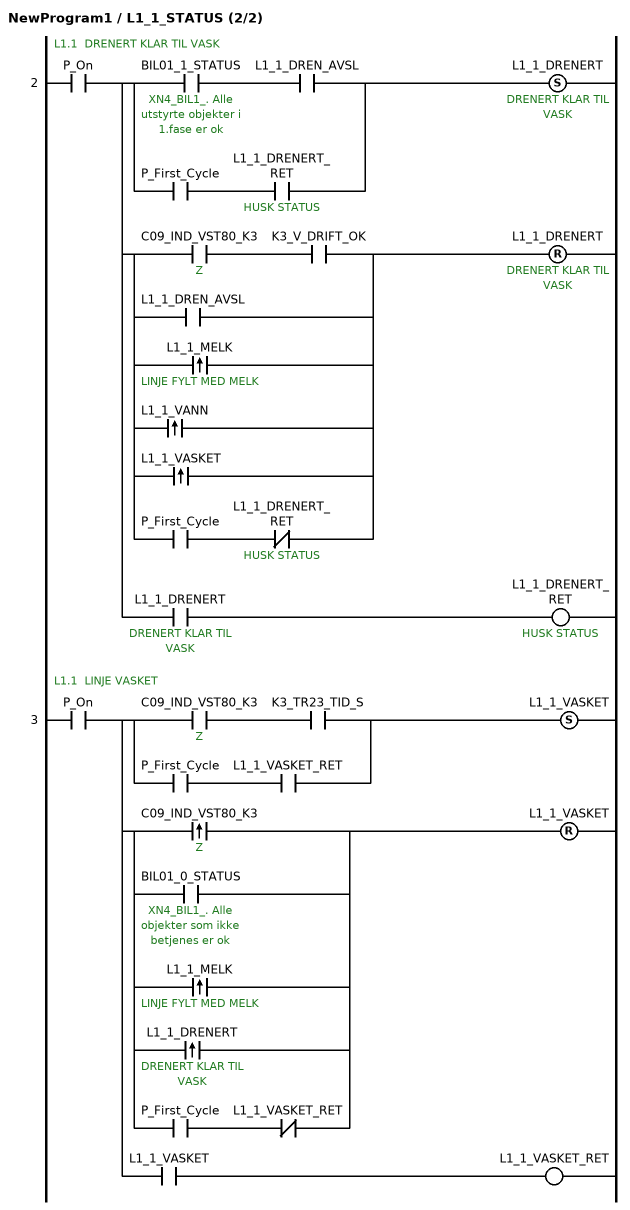
; [picture p768: NewProgram1 / L1_1_STATUS, rungs 2-3]
; rung 2: L1.1  DRENERT KLAR TIL VASK
LD P_On
OUT TR0
LD BIL01_1_STATUS  ; XN4_BIL1_. Alle utstyrte objekter i 1.fase er ok
AND L1_1_DREN_AVSL
LD P_First_Cycle
AND L1_1_DRENERT_RET  ; HUSK STATUS
ORLD
ANDLD
SET L1_1_DRENERT  ; DRENERT KLAR TIL VASK
LD TR0
LD C09_IND_VST80_K3  ; Z
AND K3_V_DRIFT_OK
OR L1_1_DREN_AVSL
@OR L1_1_MELK  ; LINJE FYLT MED MELK
@OR L1_1_VANN
@OR L1_1_VASKET
LD P_First_Cycle
ANDNOT L1_1_DRENERT_RET  ; HUSK STATUS
ORLD
ANDLD
RSET L1_1_DRENERT  ; DRENERT KLAR TIL VASK
LD TR0
AND L1_1_DRENERT  ; DRENERT KLAR TIL VASK
OUT L1_1_DRENERT_RET  ; HUSK STATUS
; rung 3: L1.1  LINJE VASKET
LD P_On
OUT TR0
LD C09_IND_VST80_K3  ; Z
AND K3_TR23_TID_S
LD P_First_Cycle
AND L1_1_VASKET_RET
ORLD
ANDLD
SET L1_1_VASKET
LD TR0
@LD C09_IND_VST80_K3  ; Z
OR BIL01_0_STATUS  ; XN4_BIL1_. Alle objekter som ikke betjenes er ok
@OR L1_1_MELK  ; LINJE FYLT MED MELK
@OR L1_1_DRENERT  ; DRENERT KLAR TIL VASK
LD P_First_Cycle
ANDNOT L1_1_VASKET_RET
ORLD
ANDLD
RSET L1_1_VASKET
LD TR0
AND L1_1_VASKET
OUT L1_1_VASKET_RET
; rung 4: Ingen_kommentar_funnet

### Section L1_1_FUNKSJONER

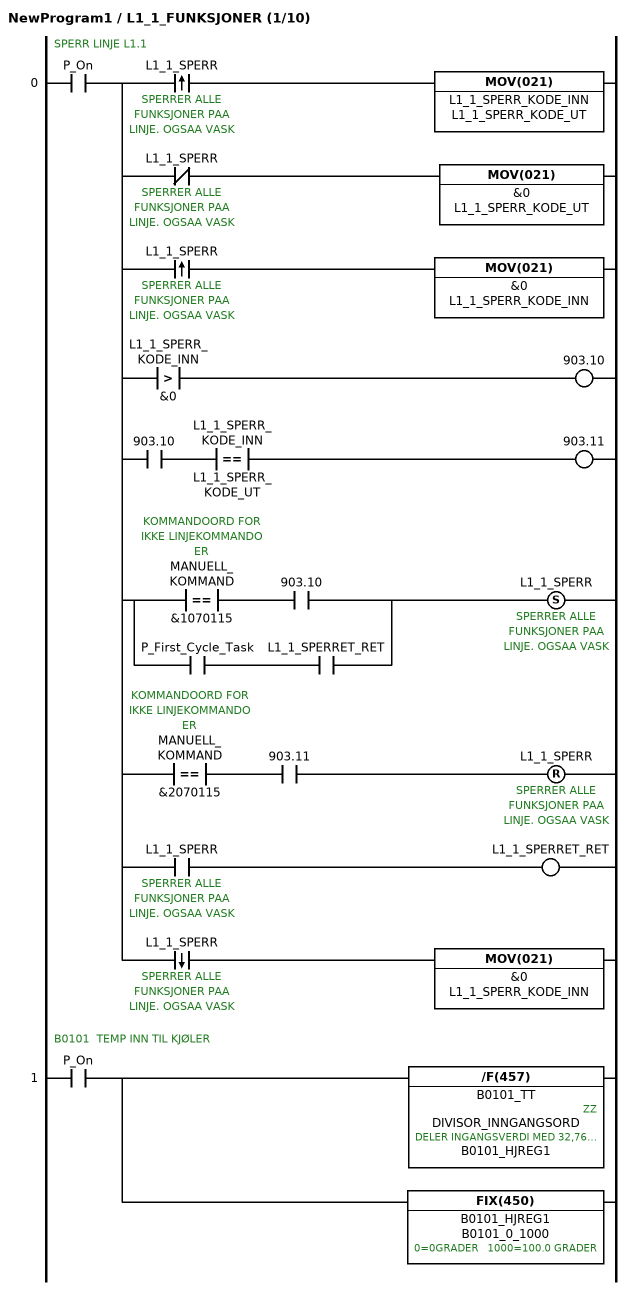
; rung 0: SPERR LINJE L1.1
LD P_On
OUT TR0
@AND L1_1_SPERR  ; SPERRER ALLE FUNKSJONER PAA LINJE. OGSAA VASK
MOV(021) L1_1_SPERR_KODE_INN L1_1_SPERR_KODE_UT
LD TR0
ANDNOT L1_1_SPERR  ; SPERRER ALLE FUNKSJONER PAA LINJE. OGSAA VASK
MOV(021) &0 L1_1_SPERR_KODE_UT
LD TR0
@AND L1_1_SPERR  ; SPERRER ALLE FUNKSJONER PAA LINJE. OGSAA VASK
MOV(021) &0 L1_1_SPERR_KODE_INN
LD TR0
AND>(320) L1_1_SPERR_KODE_INN &0
OUT 903.10
LD TR0
AND 903.10
AND=(300) L1_1_SPERR_KODE_INN L1_1_SPERR_KODE_UT
OUT 903.11
LD TR0
LD=L(301) MANUELL_KOMMAND &1070115  ; KOMMANDOORD FOR IKKE LINJEKOMMANDOER
AND 903.10
LD P_First_Cycle_Task
AND L1_1_SPERRET_RET
ORLD
ANDLD
SET L1_1_SPERR  ; SPERRER ALLE FUNKSJONER PAA LINJE. OGSAA VASK
LD TR0
AND=L(301) MANUELL_KOMMAND &2070115  ; KOMMANDOORD FOR IKKE LINJEKOMMANDOER
AND 903.11
RSET L1_1_SPERR  ; SPERRER ALLE FUNKSJONER PAA LINJE. OGSAA VASK
LD TR0
AND L1_1_SPERR  ; SPERRER ALLE FUNKSJONER PAA LINJE. OGSAA VASK
OUT L1_1_SPERRET_RET
LD TR0
%AND L1_1_SPERR  ; SPERRER ALLE FUNKSJONER PAA LINJE. OGSAA VASK
MOV(021) &0 L1_1_SPERR_KODE_INN
; rung 1: B0101  TEMP INN TIL KJØLER
LD P_On
/F(457) B0101_TT DIVISOR_INNGANGSORD B0101_HJREG1  ; ZZ, DELER INGANGSVERDI MED 32,760 FOR OMREGNING TIL 0-1000
FIX(450) B0101_HJREG1 B0101_0_1000  ; 0=0GRADER   1000=100.0 GRADER

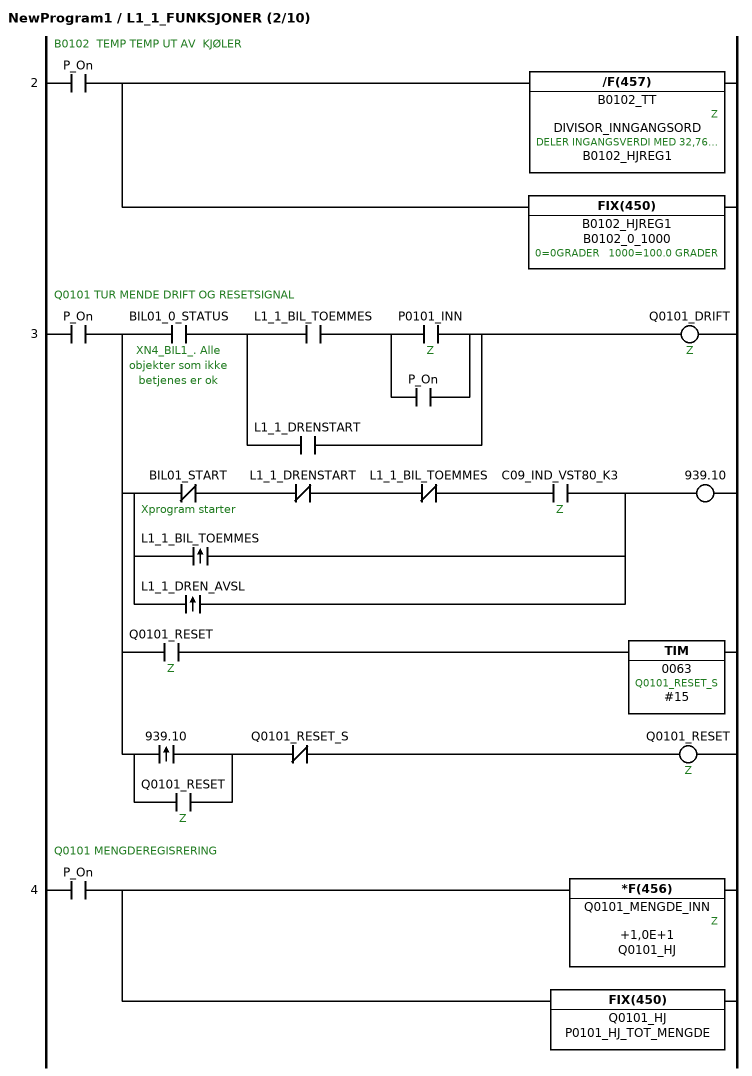
; rung 2: B0102  TEMP TEMP UT AV  KJØLER
LD P_On
/F(457) B0102_TT DIVISOR_INNGANGSORD B0102_HJREG1  ; Z, DELER INGANGSVERDI MED 32,760 FOR OMREGNING TIL 0-1000
FIX(450) B0102_HJREG1 B0102_0_1000  ; 0=0GRADER   1000=100.0 GRADER
; rung 3: Q0101 TUR MENDE DRIFT OG RESETSIGNAL
LD P_On
OUT TR0
AND BIL01_0_STATUS  ; XN4_BIL1_. Alle objekter som ikke betjenes er ok
LD L1_1_BIL_TOEMMES
LD P0101_INN  ; Z
OR P_On
ANDLD
OR L1_1_DRENSTART
ANDLD
OUT Q0101_DRIFT  ; Z
LD TR0
LDNOT BIL01_START  ; Xprogram starter
ANDNOT L1_1_DRENSTART
ANDNOT L1_1_BIL_TOEMMES
AND C09_IND_VST80_K3  ; Z
@OR L1_1_BIL_TOEMMES
@OR L1_1_DREN_AVSL
ANDLD
OUT 939.10
LD TR0
AND Q0101_RESET  ; Z
TIM 0063 #15  ; Q0101_RESET_S
LD TR0
@LD 939.10
OR Q0101_RESET  ; Z
ANDLD
ANDNOT Q0101_RESET_S
OUT Q0101_RESET  ; Z
; rung 4: Q0101 MENGDEREGISRERING
LD P_On
*F(456) Q0101_MENGDE_INN +1,0E+1 Q0101_HJ  ; Z
FIX(450) Q0101_HJ P0101_HJ_TOT_MENGDE

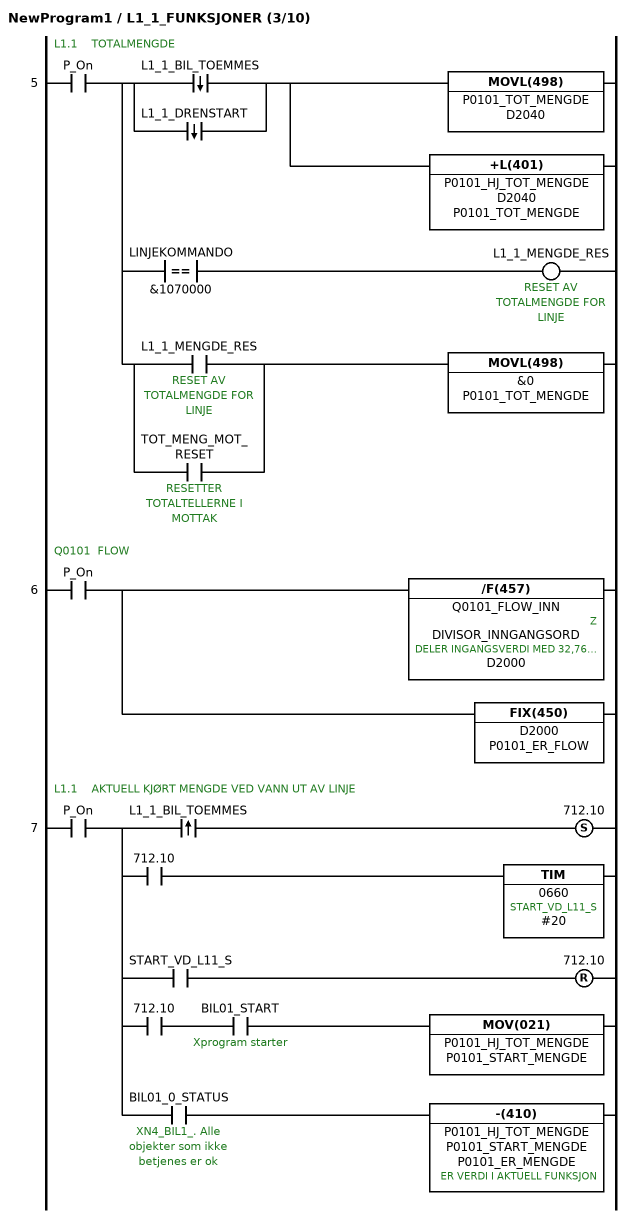
; rung 5: L1.1    TOTALMENGDE
LD P_On
OUT TR0
%LD L1_1_BIL_TOEMMES
%OR L1_1_DRENSTART
ANDLD
MOVL(498) P0101_TOT_MENGDE D2040
+L(401) P0101_HJ_TOT_MENGDE D2040 P0101_TOT_MENGDE
LD TR0
AND=L(301) LINJEKOMMANDO &1070000
OUT L1_1_MENGDE_RES  ; RESET AV  TOTALMENGDE FOR LINJE
LD TR0
LD L1_1_MENGDE_RES  ; RESET AV  TOTALMENGDE FOR LINJE
OR TOT_MENG_MOT_RESET  ; RESETTER TOTALTELLERNE I MOTTAK
ANDLD
MOVL(498) &0 P0101_TOT_MENGDE
; rung 6: Q0101  FLOW
LD P_On
/F(457) Q0101_FLOW_INN DIVISOR_INNGANGSORD D2000  ; Z, DELER INGANGSVERDI MED 32,760 FOR OMREGNING TIL 0-1000
FIX(450) D2000 P0101_ER_FLOW
; rung 7: L1.1    AKTUELL KJØRT MENGDE VED VANN UT AV LINJE
LD P_On
OUT TR0
@AND L1_1_BIL_TOEMMES
SET 712.10
LD TR0
AND 712.10
TIM 0660 #20  ; START_VD_L11_S
LD TR0
AND START_VD_L11_S
RSET 712.10
LD TR0
AND 712.10
AND BIL01_START  ; Xprogram starter
MOV(021) P0101_HJ_TOT_MENGDE P0101_START_MENGDE
LD TR0
AND BIL01_0_STATUS  ; XN4_BIL1_. Alle objekter som ikke betjenes er ok
-(410) P0101_HJ_TOT_MENGDE P0101_START_MENGDE P0101_ER_MENGDE  ; ER VERDI I AKTUELL FUNKSJON

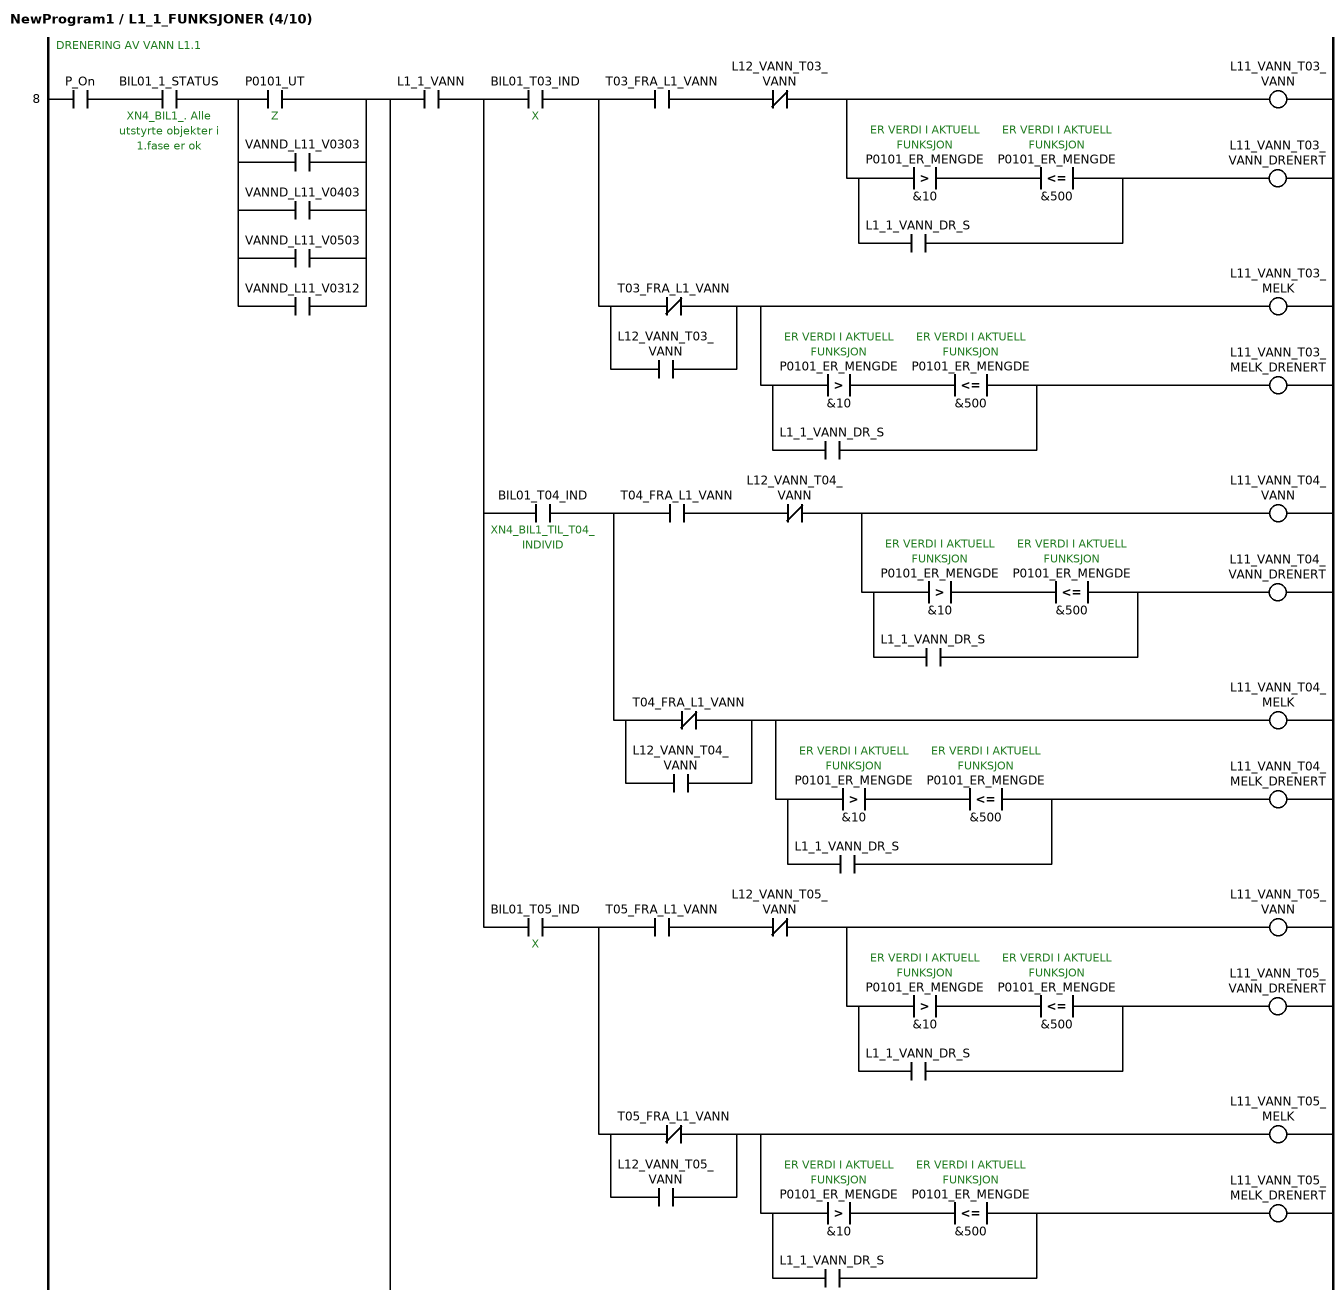

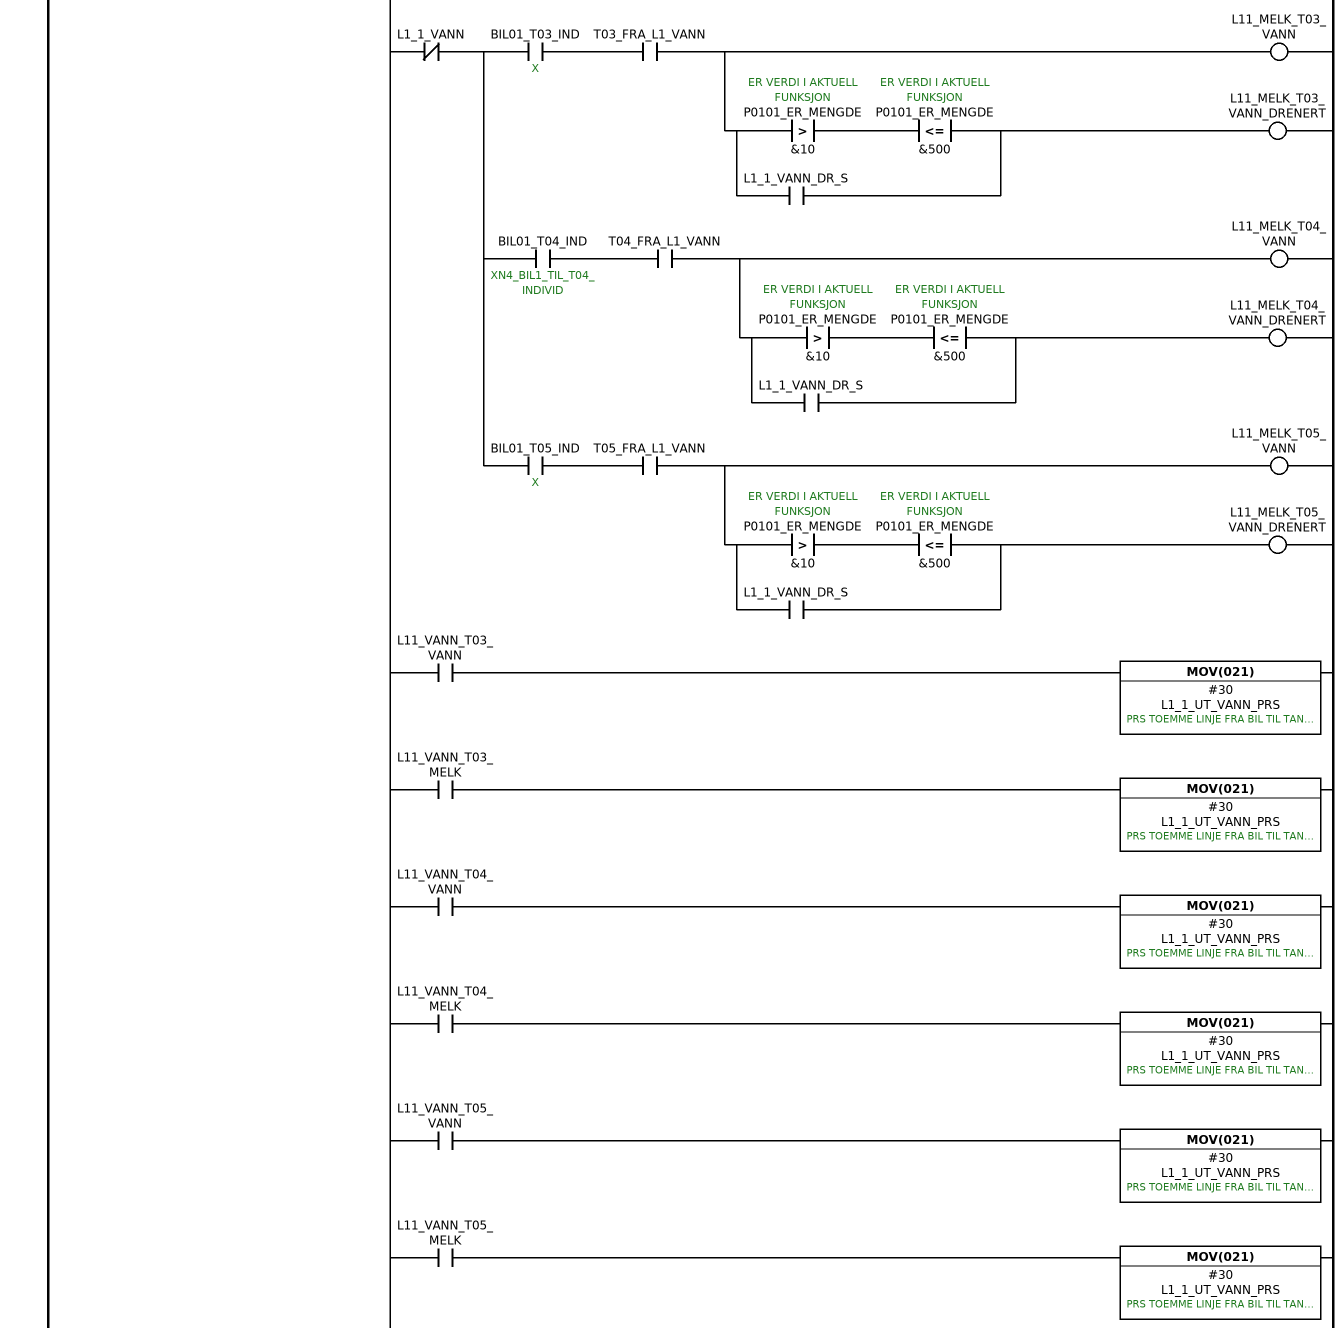

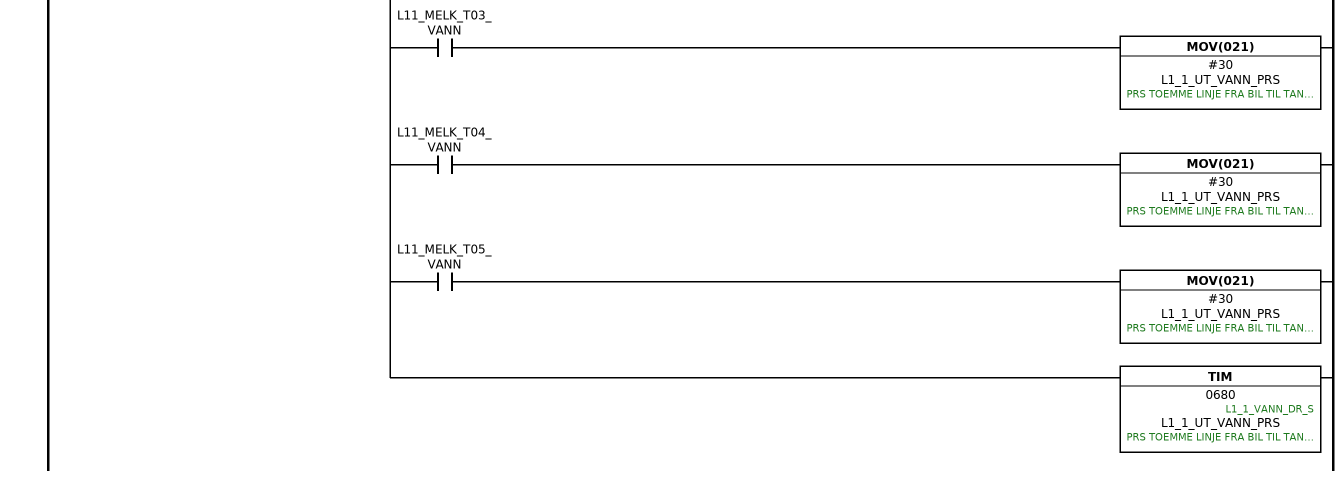
; rung 8: DRENERING AV VANN L1.1
LD P_On
AND BIL01_1_STATUS  ; XN4_BIL1_. Alle utstyrte objekter i 1.fase er ok
LD P0101_UT  ; Z
OR VANND_L11_V0303
OR VANND_L11_V0403
OR VANND_L11_V0503
OR VANND_L11_V0312
ANDLD
OUT TR0
AND L1_1_VANN
OUT TR1
AND BIL01_T03_IND  ; X
OUT TR2
AND T03_FRA_L1_VANN
ANDNOT L12_VANN_T03_VANN
OUT L11_VANN_T03_VANN
LD>(320) P0101_ER_MENGDE &10  ; ER VERDI I AKTUELL FUNKSJON
AND<=(315) P0101_ER_MENGDE &500  ; ER VERDI I AKTUELL FUNKSJON
OR L1_1_VANN_DR_S
ANDLD
OUT L11_VANN_T03_VANN_DRENERT
LD TR2
LDNOT T03_FRA_L1_VANN
OR L12_VANN_T03_VANN
ANDLD
OUT L11_VANN_T03_MELK
LD>(320) P0101_ER_MENGDE &10  ; ER VERDI I AKTUELL FUNKSJON
AND<=(315) P0101_ER_MENGDE &500  ; ER VERDI I AKTUELL FUNKSJON
OR L1_1_VANN_DR_S
ANDLD
OUT L11_VANN_T03_MELK_DRENERT
LD TR1
AND BIL01_T04_IND  ; XN4_BIL1_TIL_T04_INDIVID
OUT TR2
AND T04_FRA_L1_VANN
ANDNOT L12_VANN_T04_VANN
OUT L11_VANN_T04_VANN
LD>(320) P0101_ER_MENGDE &10  ; ER VERDI I AKTUELL FUNKSJON
AND<=(315) P0101_ER_MENGDE &500  ; ER VERDI I AKTUELL FUNKSJON
OR L1_1_VANN_DR_S
ANDLD
OUT L11_VANN_T04_VANN_DRENERT
LD TR2
LDNOT T04_FRA_L1_VANN
OR L12_VANN_T04_VANN
ANDLD
OUT L11_VANN_T04_MELK
LD>(320) P0101_ER_MENGDE &10  ; ER VERDI I AKTUELL FUNKSJON
AND<=(315) P0101_ER_MENGDE &500  ; ER VERDI I AKTUELL FUNKSJON
OR L1_1_VANN_DR_S
ANDLD
OUT L11_VANN_T04_MELK_DRENERT
LD TR1
AND BIL01_T05_IND  ; X
OUT TR1
AND T05_FRA_L1_VANN
ANDNOT L12_VANN_T05_VANN
OUT L11_VANN_T05_VANN
LD>(320) P0101_ER_MENGDE &10  ; ER VERDI I AKTUELL FUNKSJON
AND<=(315) P0101_ER_MENGDE &500  ; ER VERDI I AKTUELL FUNKSJON
OR L1_1_VANN_DR_S
ANDLD
OUT L11_VANN_T05_VANN_DRENERT
LD TR1
LDNOT T05_FRA_L1_VANN
OR L12_VANN_T05_VANN
ANDLD
OUT L11_VANN_T05_MELK
LD>(320) P0101_ER_MENGDE &10  ; ER VERDI I AKTUELL FUNKSJON
AND<=(315) P0101_ER_MENGDE &500  ; ER VERDI I AKTUELL FUNKSJON
OR L1_1_VANN_DR_S
ANDLD
OUT L11_VANN_T05_MELK_DRENERT
LD TR0
ANDNOT L1_1_VANN
OUT TR1
AND BIL01_T03_IND  ; X
AND T03_FRA_L1_VANN
OUT L11_MELK_T03_VANN
LD>(320) P0101_ER_MENGDE &10  ; ER VERDI I AKTUELL FUNKSJON
AND<=(315) P0101_ER_MENGDE &500  ; ER VERDI I AKTUELL FUNKSJON
OR L1_1_VANN_DR_S
ANDLD
OUT L11_MELK_T03_VANN_DRENERT
LD TR1
AND BIL01_T04_IND  ; XN4_BIL1_TIL_T04_INDIVID
AND T04_FRA_L1_VANN
OUT L11_MELK_T04_VANN
LD>(320) P0101_ER_MENGDE &10  ; ER VERDI I AKTUELL FUNKSJON
AND<=(315) P0101_ER_MENGDE &500  ; ER VERDI I AKTUELL FUNKSJON
OR L1_1_VANN_DR_S
ANDLD
OUT L11_MELK_T04_VANN_DRENERT
LD TR1
AND BIL01_T05_IND  ; X
AND T05_FRA_L1_VANN
OUT L11_MELK_T05_VANN
LD>(320) P0101_ER_MENGDE &10  ; ER VERDI I AKTUELL FUNKSJON
AND<=(315) P0101_ER_MENGDE &500  ; ER VERDI I AKTUELL FUNKSJON
OR L1_1_VANN_DR_S
ANDLD
OUT L11_MELK_T05_VANN_DRENERT
LD TR0
AND L11_VANN_T03_VANN
MOV(021) #30 L1_1_UT_VANN_PRS  ; PRS TOEMME LINJE FRA BIL TIL TANK FOR VANN
LD TR0
AND L11_VANN_T03_MELK
MOV(021) #30 L1_1_UT_VANN_PRS  ; PRS TOEMME LINJE FRA BIL TIL TANK FOR VANN
LD TR0
AND L11_VANN_T04_VANN
MOV(021) #30 L1_1_UT_VANN_PRS  ; PRS TOEMME LINJE FRA BIL TIL TANK FOR VANN
LD TR0
AND L11_VANN_T04_MELK
MOV(021) #30 L1_1_UT_VANN_PRS  ; PRS TOEMME LINJE FRA BIL TIL TANK FOR VANN
LD TR0
AND L11_VANN_T05_VANN
MOV(021) #30 L1_1_UT_VANN_PRS  ; PRS TOEMME LINJE FRA BIL TIL TANK FOR VANN
LD TR0
AND L11_VANN_T05_MELK
MOV(021) #30 L1_1_UT_VANN_PRS  ; PRS TOEMME LINJE FRA BIL TIL TANK FOR VANN
LD TR0
AND L11_MELK_T03_VANN
MOV(021) #30 L1_1_UT_VANN_PRS  ; PRS TOEMME LINJE FRA BIL TIL TANK FOR VANN
LD TR0
AND L11_MELK_T04_VANN
MOV(021) #30 L1_1_UT_VANN_PRS  ; PRS TOEMME LINJE FRA BIL TIL TANK FOR VANN
LD TR0
AND L11_MELK_T05_VANN
MOV(021) #30 L1_1_UT_VANN_PRS  ; PRS TOEMME LINJE FRA BIL TIL TANK FOR VANN
LD TR0
TIM 0680 L1_1_UT_VANN_PRS  ; PRS TOEMME LINJE FRA BIL TIL TANK FOR VANN, L1_1_VANN_DR_S

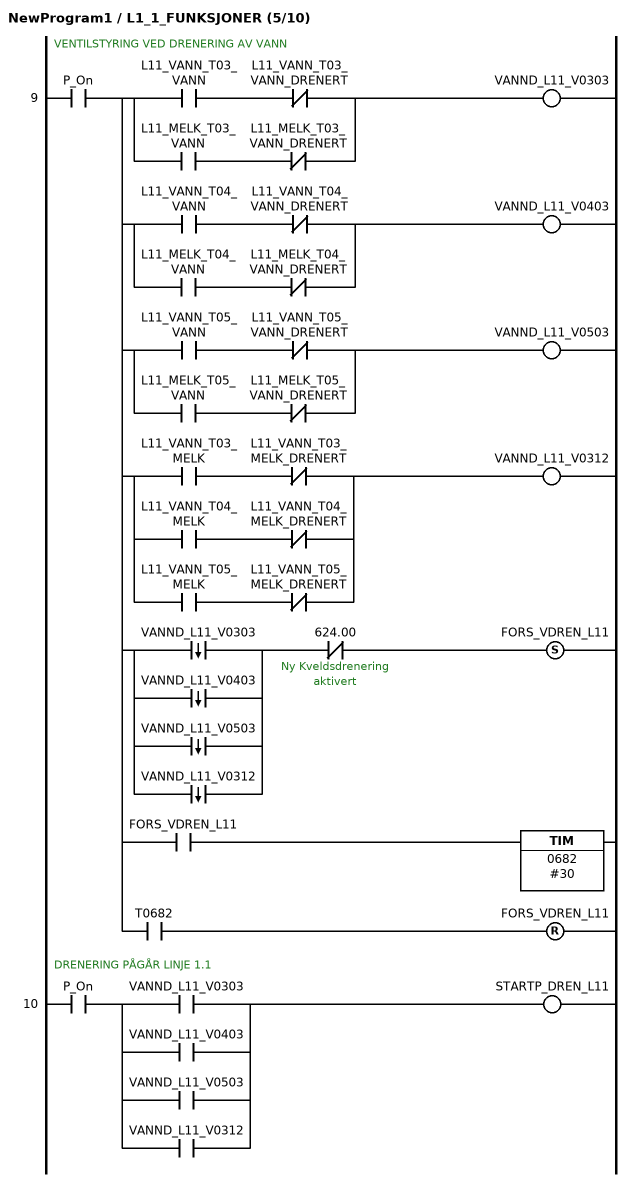
; rung 9: VENTILSTYRING VED DRENERING AV VANN
LD P_On
OUT TR0
LD L11_VANN_T03_VANN
ANDNOT L11_VANN_T03_VANN_DRENERT
LD L11_MELK_T03_VANN
ANDNOT L11_MELK_T03_VANN_DRENERT
ORLD
ANDLD
OUT VANND_L11_V0303
LD TR0
LD L11_VANN_T04_VANN
ANDNOT L11_VANN_T04_VANN_DRENERT
LD L11_MELK_T04_VANN
ANDNOT L11_MELK_T04_VANN_DRENERT
ORLD
ANDLD
OUT VANND_L11_V0403
LD TR0
LD L11_VANN_T05_VANN
ANDNOT L11_VANN_T05_VANN_DRENERT
LD L11_MELK_T05_VANN
ANDNOT L11_MELK_T05_VANN_DRENERT
ORLD
ANDLD
OUT VANND_L11_V0503
LD TR0
LD L11_VANN_T03_MELK
ANDNOT L11_VANN_T03_MELK_DRENERT
LD L11_VANN_T04_MELK
ANDNOT L11_VANN_T04_MELK_DRENERT
ORLD
LD L11_VANN_T05_MELK
ANDNOT L11_VANN_T05_MELK_DRENERT
ORLD
ANDLD
OUT VANND_L11_V0312
LD TR0
%LD VANND_L11_V0303
%OR VANND_L11_V0403
%OR VANND_L11_V0503
%OR VANND_L11_V0312
ANDLD
ANDNOT 624.00  ; Ny Kveldsdrenering aktivert
SET FORS_VDREN_L11
LD TR0
AND FORS_VDREN_L11
TIM 0682 #30
LD TR0
AND T0682
RSET FORS_VDREN_L11
; rung 10: DRENERING PÅGÅR LINJE 1.1
LD P_On
LD VANND_L11_V0303
OR VANND_L11_V0403
OR VANND_L11_V0503
OR VANND_L11_V0312
ANDLD
OUT STARTP_DREN_L11

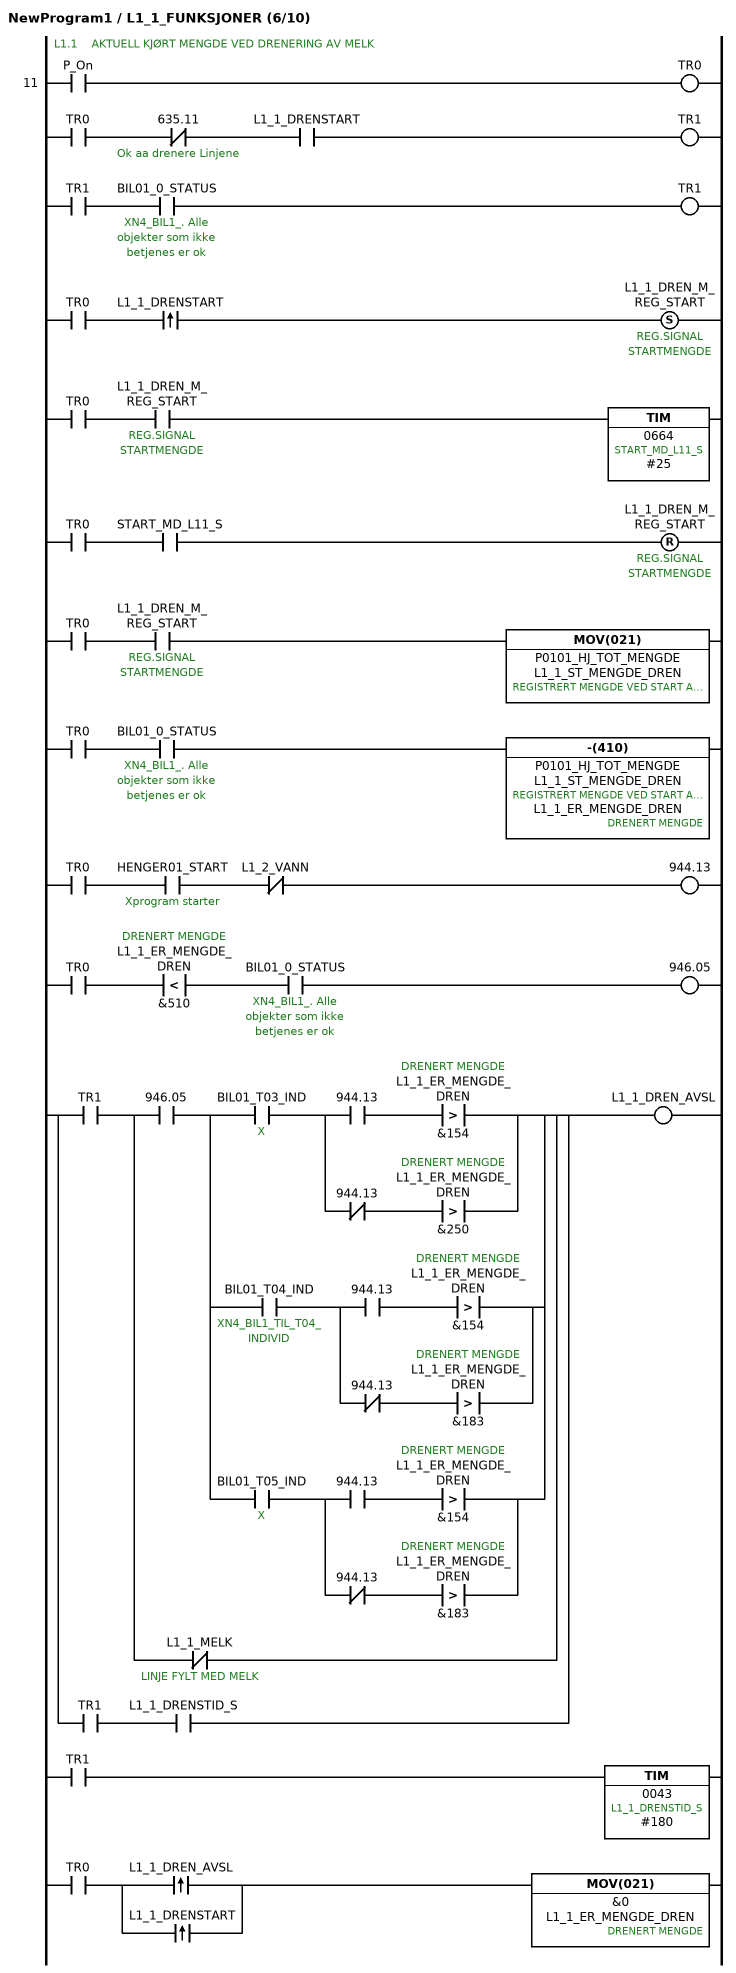
; rung 11: L1.1    AKTUELL KJØRT MENGDE VED DRENERING AV MELK
LD P_On
OUT TR0
@AND L1_1_DRENSTART
SET L1_1_DREN_M_REG_START  ; REG.SIGNAL STARTMENGDE
LD TR0
AND L1_1_DREN_M_REG_START  ; REG.SIGNAL STARTMENGDE
TIM 0664 #25  ; START_MD_L11_S
LD TR0
AND START_MD_L11_S
RSET L1_1_DREN_M_REG_START  ; REG.SIGNAL STARTMENGDE
LD TR0
AND L1_1_DREN_M_REG_START  ; REG.SIGNAL STARTMENGDE
MOV(021) P0101_HJ_TOT_MENGDE L1_1_ST_MENGDE_DREN  ; REGISTRERT MENGDE VED START AV DREN.
LD TR0
AND BIL01_0_STATUS  ; XN4_BIL1_. Alle objekter som ikke betjenes er ok
-(410) P0101_HJ_TOT_MENGDE L1_1_ST_MENGDE_DREN L1_1_ER_MENGDE_DREN  ; REGISTRERT MENGDE VED START AV DREN., DRENERT MENGDE
LD TR0
AND HENGER01_START  ; Xprogram starter
ANDNOT L1_2_VANN
OUT 944.13
LD TR0
AND<(310) L1_1_ER_MENGDE_DREN &510  ; DRENERT MENGDE
AND BIL01_0_STATUS  ; XN4_BIL1_. Alle objekter som ikke betjenes er ok
OUT 946.05
LD TR0
ANDNOT 635.11  ; Ok aa drenere Linjene
AND L1_1_DRENSTART
OUT TR1
LD 946.05
LD BIL01_T03_IND  ; X
LD 944.13
AND>(320) L1_1_ER_MENGDE_DREN &154  ; DRENERT MENGDE
LDNOT 944.13
AND>(320) L1_1_ER_MENGDE_DREN &250  ; DRENERT MENGDE
ORLD
ANDLD
LD BIL01_T04_IND  ; XN4_BIL1_TIL_T04_INDIVID
LD 944.13
AND>(320) L1_1_ER_MENGDE_DREN &154  ; DRENERT MENGDE
LDNOT 944.13
AND>(320) L1_1_ER_MENGDE_DREN &183  ; DRENERT MENGDE
ORLD
ANDLD
ORLD
LD BIL01_T05_IND  ; X
LD 944.13
AND>(320) L1_1_ER_MENGDE_DREN &154  ; DRENERT MENGDE
LDNOT 944.13
AND>(320) L1_1_ER_MENGDE_DREN &183  ; DRENERT MENGDE
ORLD
ANDLD
ORLD
ANDLD
ORNOT L1_1_MELK  ; LINJE FYLT MED MELK
ANDLD
LD TR1
AND BIL01_0_STATUS  ; XN4_BIL1_. Alle objekter som ikke betjenes er ok
OUT TR1
AND L1_1_DRENSTID_S
ORLD
OUT L1_1_DREN_AVSL
LD TR1
TIM 0043 #180  ; L1_1_DRENSTID_S
LD TR0
@LD L1_1_DREN_AVSL
@OR L1_1_DRENSTART
ANDLD
MOV(021) &0 L1_1_ER_MENGDE_DREN  ; DRENERT MENGDE

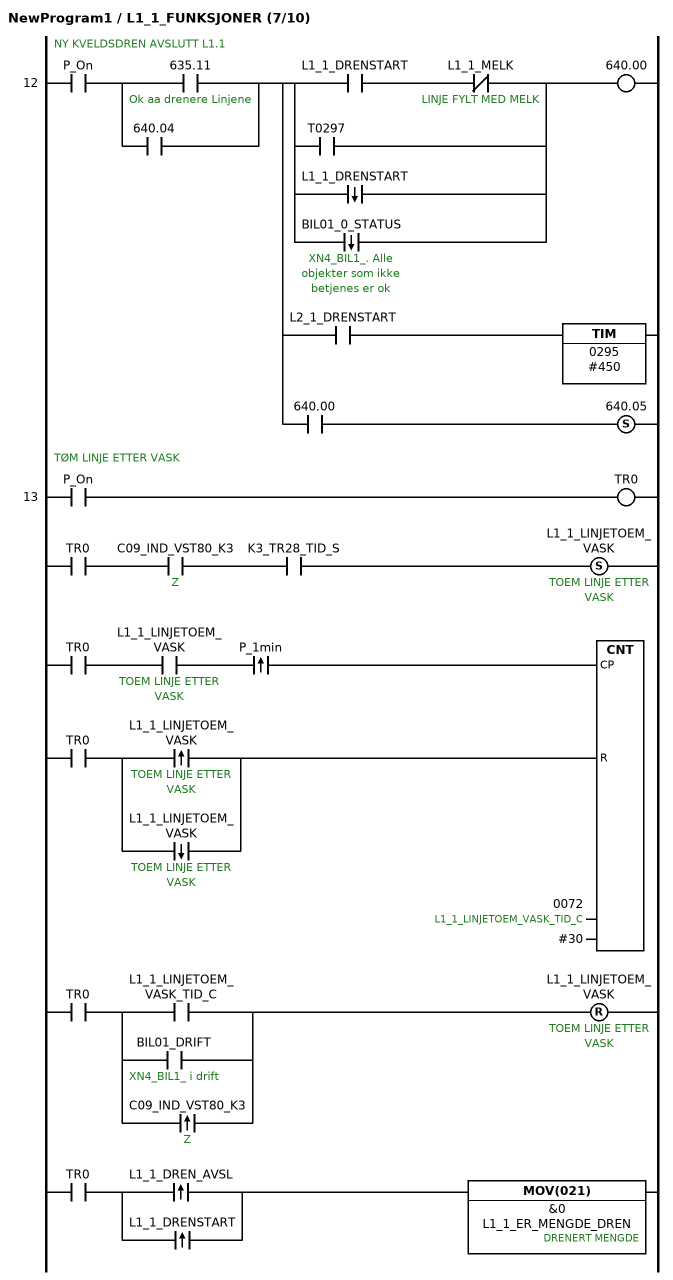
; rung 12: NY KVELDSDREN AVSLUTT L1.1
LD P_On
LD 635.11  ; Ok aa drenere Linjene
OR 640.04
ANDLD
OUT TR0
LD L1_1_DRENSTART
ANDNOT L1_1_MELK  ; LINJE FYLT MED MELK
OR T0297
%OR L1_1_DRENSTART
%OR BIL01_0_STATUS  ; XN4_BIL1_. Alle objekter som ikke betjenes er ok
ANDLD
OUT 640.00
LD TR0
AND L2_1_DRENSTART
TIM 0295 #450
LD TR0
AND 640.00
SET 640.05
; rung 13: TØM LINJE ETTER VASK
LD P_On
OUT TR0
AND C09_IND_VST80_K3  ; Z
AND K3_TR28_TID_S
SET L1_1_LINJETOEM_VASK  ; TOEM LINJE ETTER VASK
LD TR0
AND L1_1_LINJETOEM_VASK  ; TOEM LINJE ETTER VASK
@AND P_1min
LD TR0
@LD L1_1_LINJETOEM_VASK  ; TOEM LINJE ETTER VASK
%OR L1_1_LINJETOEM_VASK  ; TOEM LINJE ETTER VASK
ANDLD
CNT 0072 #30  ; L1_1_LINJETOEM_VASK_TID_C
LD TR0
LD L1_1_LINJETOEM_VASK_TID_C
OR BIL01_DRIFT  ; XN4_BIL1_ i drift
@OR C09_IND_VST80_K3  ; Z
ANDLD
RSET L1_1_LINJETOEM_VASK  ; TOEM LINJE ETTER VASK
LD TR0
@LD L1_1_DREN_AVSL
@OR L1_1_DRENSTART
ANDLD
MOV(021) &0 L1_1_ER_MENGDE_DREN  ; DRENERT MENGDE

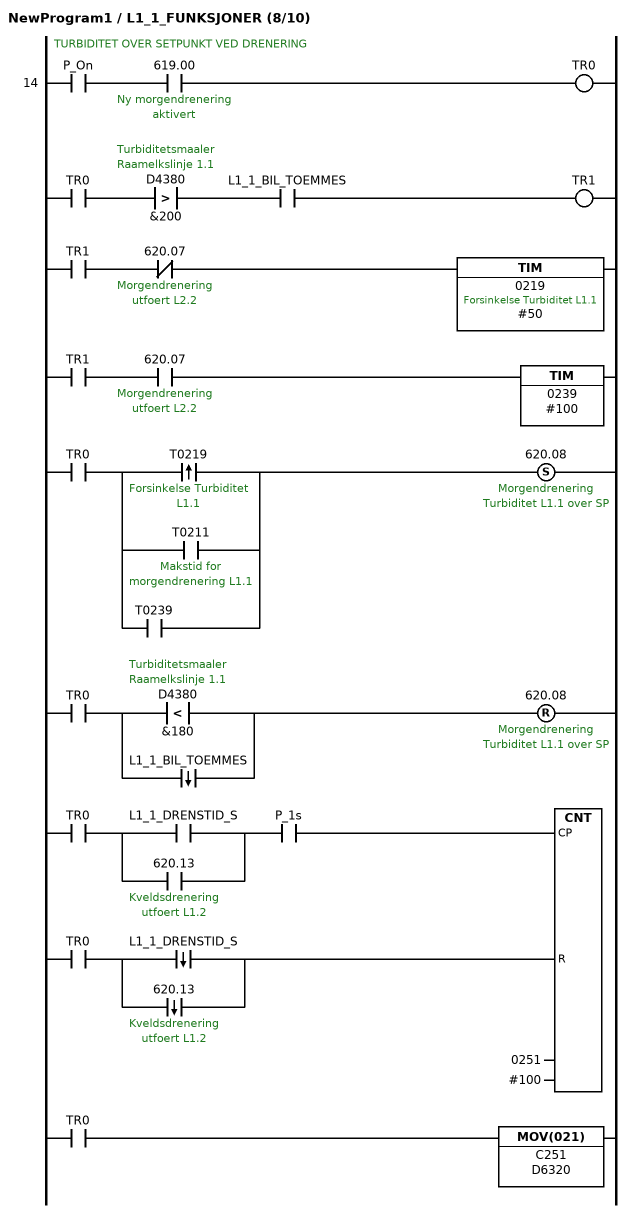
; rung 14: TURBIDITET OVER SETPUNKT VED DRENERING
LD P_On
AND 619.00  ; Ny morgendrenering aktivert
OUT TR0
AND>(320) D4380 &200  ; Turbiditetsmaaler Raamelkslinje 1.1
AND L1_1_BIL_TOEMMES
OUT TR1
ANDNOT 620.07  ; Morgendrenering utfoert L2.2
TIM 0219 #50  ; Forsinkelse Turbiditet L1.1
LD TR1
AND 620.07  ; Morgendrenering utfoert L2.2
TIM 0239 #100
LD TR0
@LD T0219  ; Forsinkelse Turbiditet L1.1
OR T0211  ; Makstid for morgendrenering L1.1
OR T0239
ANDLD
SET 620.08  ; Morgendrenering Turbiditet L1.1 over SP
LD TR0
LD<(310) D4380 &180  ; Turbiditetsmaaler Raamelkslinje 1.1
%OR L1_1_BIL_TOEMMES
ANDLD
RSET 620.08  ; Morgendrenering Turbiditet L1.1 over SP
LD TR0
LD L1_1_DRENSTID_S
OR 620.13  ; Kveldsdrenering utfoert L1.2
ANDLD
AND P_1s
LD TR0
%LD L1_1_DRENSTID_S
%OR 620.13  ; Kveldsdrenering utfoert L1.2
ANDLD
CNT 0251 #100
LD TR0
MOV(021) C251 D6320

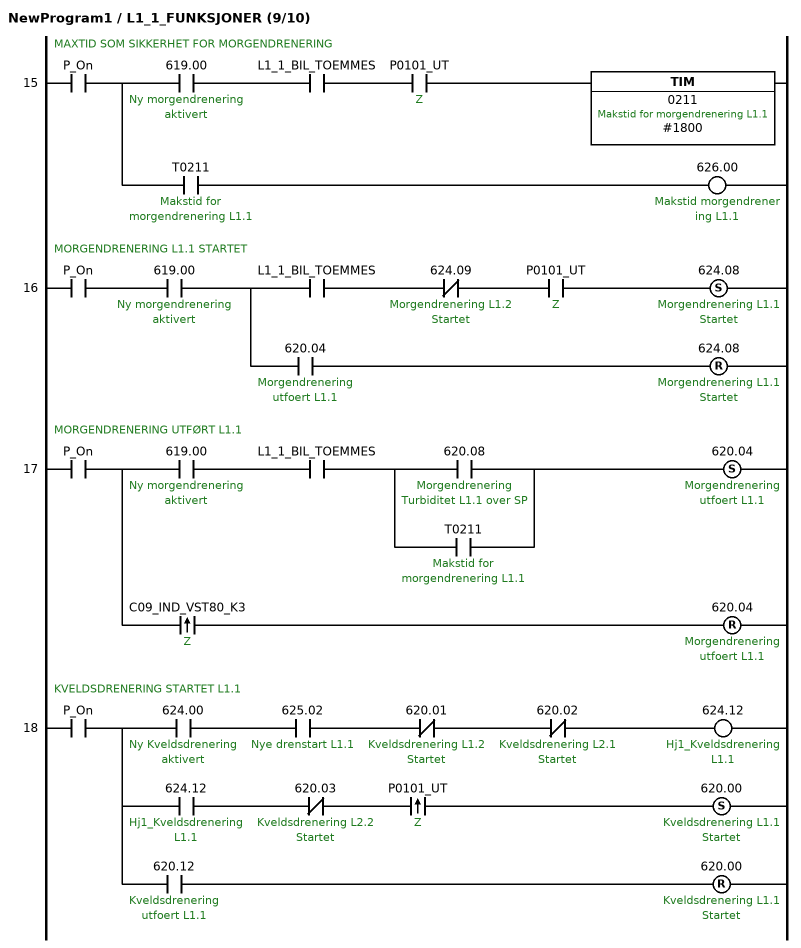
; rung 15: MAXTID SOM SIKKERHET FOR MORGENDRENERING
LD P_On
OUT TR0
AND 619.00  ; Ny morgendrenering aktivert
AND L1_1_BIL_TOEMMES
AND P0101_UT  ; Z
TIM 0211 #1800  ; Makstid for morgendrenering L1.1
LD TR0
AND T0211  ; Makstid for morgendrenering L1.1
OUT 626.00  ; Makstid morgendrenering L1.1
; rung 16: MORGENDRENERING L1.1 STARTET
LD P_On
AND 619.00  ; Ny morgendrenering aktivert
OUT TR0
AND L1_1_BIL_TOEMMES
ANDNOT 624.09  ; Morgendrenering L1.2 Startet
AND P0101_UT  ; Z
SET 624.08  ; Morgendrenering L1.1 Startet
LD TR0
AND 620.04  ; Morgendrenering utfoert L1.1
RSET 624.08  ; Morgendrenering L1.1 Startet
; rung 17: MORGENDRENERING UTFØRT L1.1
LD P_On
OUT TR0
AND 619.00  ; Ny morgendrenering aktivert
AND L1_1_BIL_TOEMMES
LD 620.08  ; Morgendrenering Turbiditet L1.1 over SP
OR T0211  ; Makstid for morgendrenering L1.1
ANDLD
SET 620.04  ; Morgendrenering utfoert L1.1
LD TR0
@AND C09_IND_VST80_K3  ; Z
RSET 620.04  ; Morgendrenering utfoert L1.1
; rung 18: KVELDSDRENERING STARTET L1.1
LD P_On
OUT TR0
AND 624.00  ; Ny Kveldsdrenering aktivert
AND 625.02  ; Nye drenstart L1.1
ANDNOT 620.01  ; Kveldsdrenering L1.2 Startet
ANDNOT 620.02  ; Kveldsdrenering L2.1 Startet
OUT 624.12  ; Hj1_Kveldsdrenering L1.1
LD TR0
AND 624.12  ; Hj1_Kveldsdrenering L1.1
ANDNOT 620.03  ; Kveldsdrenering L2.2 Startet
@AND P0101_UT  ; Z
SET 620.00  ; Kveldsdrenering L1.1 Startet
LD TR0
AND 620.12  ; Kveldsdrenering utfoert L1.1
RSET 620.00  ; Kveldsdrenering L1.1 Startet

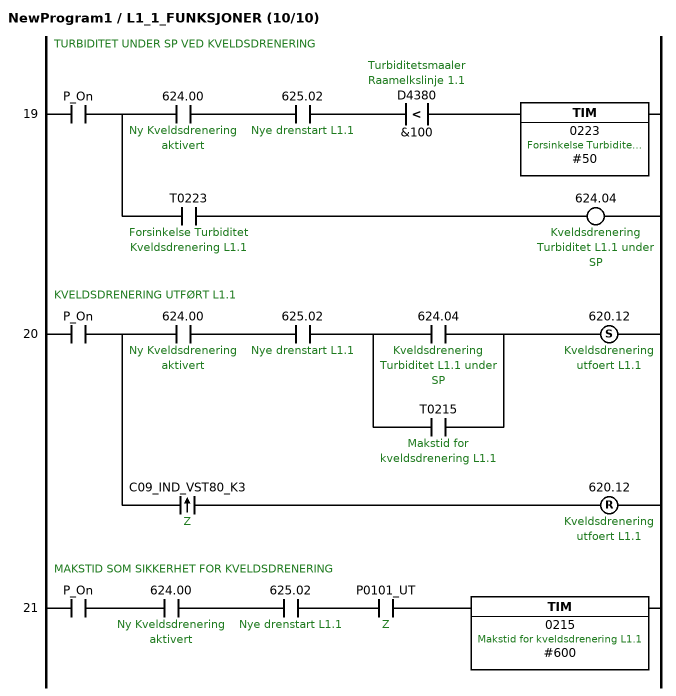
; rung 19: TURBIDITET UNDER SP VED KVELDSDRENERING
LD P_On
OUT TR0
AND 624.00  ; Ny Kveldsdrenering aktivert
AND 625.02  ; Nye drenstart L1.1
AND<(310) D4380 &100  ; Turbiditetsmaaler Raamelkslinje 1.1
TIM 0223 #50  ; Forsinkelse Turbiditet Kveldsdrenering L1.1
LD TR0
AND T0223  ; Forsinkelse Turbiditet Kveldsdrenering L1.1
OUT 624.04  ; Kveldsdrenering Turbiditet L1.1 under SP
; rung 20: KVELDSDRENERING UTFØRT L1.1
LD P_On
OUT TR0
AND 624.00  ; Ny Kveldsdrenering aktivert
AND 625.02  ; Nye drenstart L1.1
LD 624.04  ; Kveldsdrenering Turbiditet L1.1 under SP
OR T0215  ; Makstid for kveldsdrenering L1.1
ANDLD
SET 620.12  ; Kveldsdrenering utfoert L1.1
LD TR0
@AND C09_IND_VST80_K3  ; Z
RSET 620.12  ; Kveldsdrenering utfoert L1.1
; rung 21: MAKSTID SOM SIKKERHET FOR KVELDSDRENERING
LD P_On
AND 624.00  ; Ny Kveldsdrenering aktivert
AND 625.02  ; Nye drenstart L1.1
AND P0101_UT  ; Z
TIM 0215 #600  ; Makstid for kveldsdrenering L1.1
; rung 22: Ingen_kommentar_funnet

### Section L1_2_STATUS

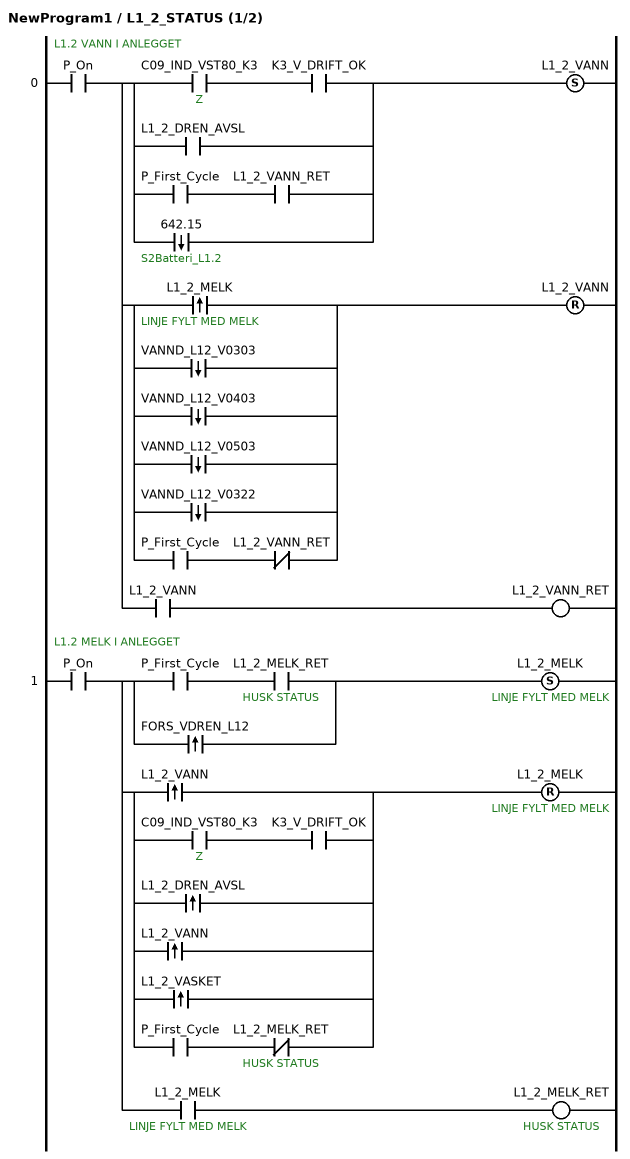
; rung 0: L1.2 VANN I ANLEGGET
LD P_On
OUT TR0
LD C09_IND_VST80_K3  ; Z
AND K3_V_DRIFT_OK
OR L1_2_DREN_AVSL
LD P_First_Cycle
AND L1_2_VANN_RET
ORLD
%OR 642.15  ; S2Batteri_L1.2
ANDLD
SET L1_2_VANN
LD TR0
@LD L1_2_MELK  ; LINJE FYLT MED MELK
%OR VANND_L12_V0303
%OR VANND_L12_V0403
%OR VANND_L12_V0503
%OR VANND_L12_V0322
LD P_First_Cycle
ANDNOT L1_2_VANN_RET
ORLD
ANDLD
RSET L1_2_VANN
LD TR0
AND L1_2_VANN
OUT L1_2_VANN_RET
; rung 1: L1.2 MELK I ANLEGGET
LD P_On
OUT TR0
LD P_First_Cycle
AND L1_2_MELK_RET  ; HUSK STATUS
@OR FORS_VDREN_L12
ANDLD
SET L1_2_MELK  ; LINJE FYLT MED MELK
LD TR0
@LD L1_2_VANN
LD C09_IND_VST80_K3  ; Z
AND K3_V_DRIFT_OK
ORLD
@OR L1_2_DREN_AVSL
@OR L1_2_VANN
@OR L1_2_VASKET
LD P_First_Cycle
ANDNOT L1_2_MELK_RET  ; HUSK STATUS
ORLD
ANDLD
RSET L1_2_MELK  ; LINJE FYLT MED MELK
LD TR0
AND L1_2_MELK  ; LINJE FYLT MED MELK
OUT L1_2_MELK_RET  ; HUSK STATUS

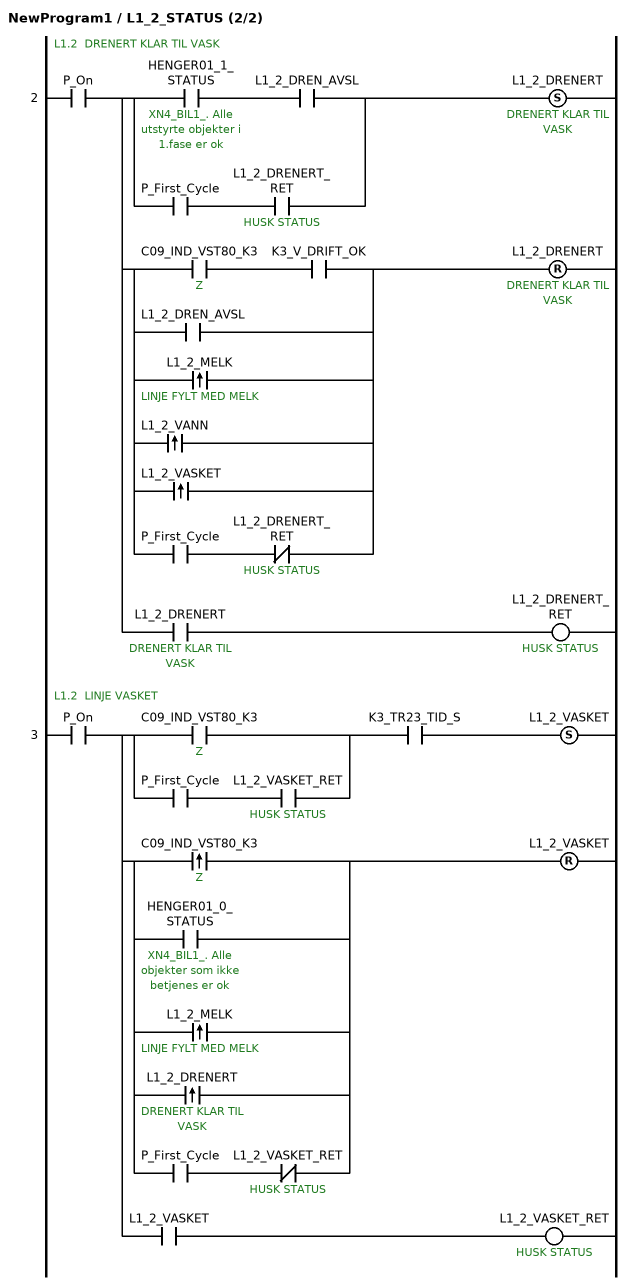
; rung 2: L1.2  DRENERT KLAR TIL VASK
LD P_On
OUT TR0
LD HENGER01_1_STATUS  ; XN4_BIL1_. Alle utstyrte objekter i 1.fase er ok
AND L1_2_DREN_AVSL
LD P_First_Cycle
AND L1_2_DRENERT_RET  ; HUSK STATUS
ORLD
ANDLD
SET L1_2_DRENERT  ; DRENERT KLAR TIL VASK
LD TR0
LD C09_IND_VST80_K3  ; Z
AND K3_V_DRIFT_OK
OR L1_2_DREN_AVSL
@OR L1_2_MELK  ; LINJE FYLT MED MELK
@OR L1_2_VANN
@OR L1_2_VASKET
LD P_First_Cycle
ANDNOT L1_2_DRENERT_RET  ; HUSK STATUS
ORLD
ANDLD
RSET L1_2_DRENERT  ; DRENERT KLAR TIL VASK
LD TR0
AND L1_2_DRENERT  ; DRENERT KLAR TIL VASK
OUT L1_2_DRENERT_RET  ; HUSK STATUS
; rung 3: L1.2  LINJE VASKET
LD P_On
OUT TR0
LD C09_IND_VST80_K3  ; Z
LD P_First_Cycle
AND L1_2_VASKET_RET  ; HUSK STATUS
ORLD
ANDLD
AND K3_TR23_TID_S
SET L1_2_VASKET
LD TR0
@LD C09_IND_VST80_K3  ; Z
OR HENGER01_0_STATUS  ; XN4_BIL1_. Alle objekter som ikke betjenes er ok
@OR L1_2_MELK  ; LINJE FYLT MED MELK
@OR L1_2_DRENERT  ; DRENERT KLAR TIL VASK
LD P_First_Cycle
ANDNOT L1_2_VASKET_RET  ; HUSK STATUS
ORLD
ANDLD
RSET L1_2_VASKET
LD TR0
AND L1_2_VASKET
OUT L1_2_VASKET_RET  ; HUSK STATUS
; rung 4: Ingen_kommentar_funnet

### Section L1_2_FUNKSJONER

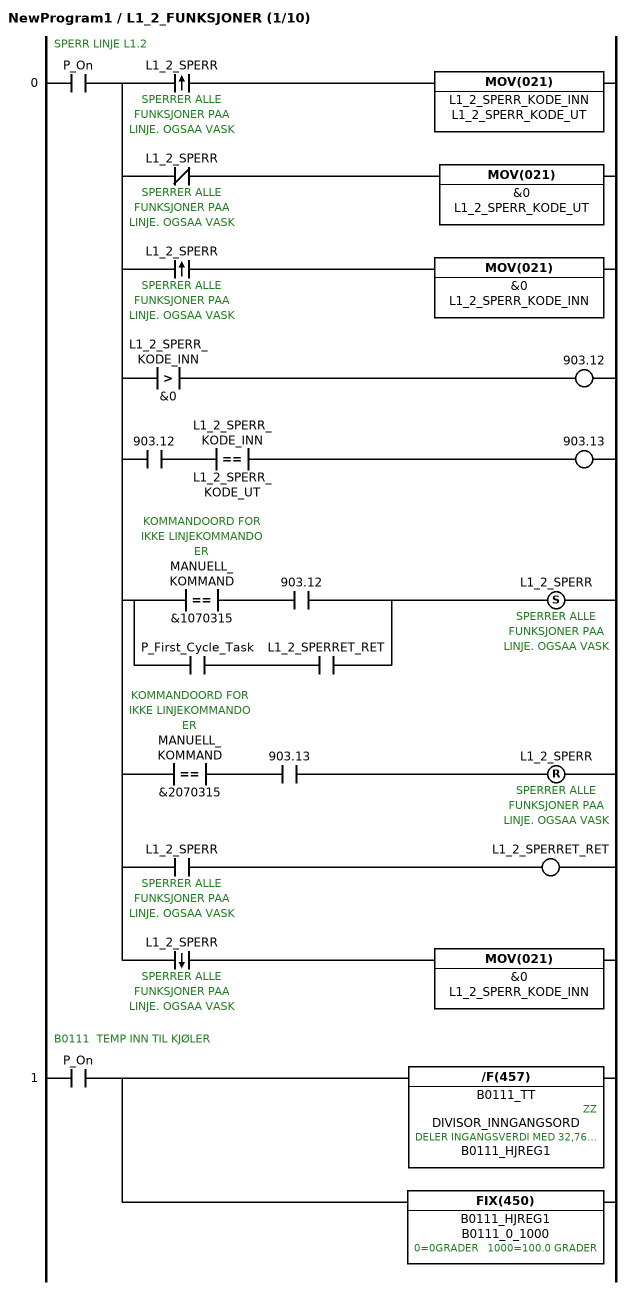
; rung 0: SPERR LINJE L1.2
LD P_On
OUT TR0
@AND L1_2_SPERR  ; SPERRER ALLE FUNKSJONER PAA LINJE. OGSAA VASK
MOV(021) L1_2_SPERR_KODE_INN L1_2_SPERR_KODE_UT
LD TR0
ANDNOT L1_2_SPERR  ; SPERRER ALLE FUNKSJONER PAA LINJE. OGSAA VASK
MOV(021) &0 L1_2_SPERR_KODE_UT
LD TR0
@AND L1_2_SPERR  ; SPERRER ALLE FUNKSJONER PAA LINJE. OGSAA VASK
MOV(021) &0 L1_2_SPERR_KODE_INN
LD TR0
AND>(320) L1_2_SPERR_KODE_INN &0
OUT 903.12
LD TR0
AND 903.12
AND=(300) L1_2_SPERR_KODE_INN L1_2_SPERR_KODE_UT
OUT 903.13
LD TR0
LD=L(301) MANUELL_KOMMAND &1070315  ; KOMMANDOORD FOR IKKE LINJEKOMMANDOER
AND 903.12
LD P_First_Cycle_Task
AND L1_2_SPERRET_RET
ORLD
ANDLD
SET L1_2_SPERR  ; SPERRER ALLE FUNKSJONER PAA LINJE. OGSAA VASK
LD TR0
AND=L(301) MANUELL_KOMMAND &2070315  ; KOMMANDOORD FOR IKKE LINJEKOMMANDOER
AND 903.13
RSET L1_2_SPERR  ; SPERRER ALLE FUNKSJONER PAA LINJE. OGSAA VASK
LD TR0
AND L1_2_SPERR  ; SPERRER ALLE FUNKSJONER PAA LINJE. OGSAA VASK
OUT L1_2_SPERRET_RET
LD TR0
%AND L1_2_SPERR  ; SPERRER ALLE FUNKSJONER PAA LINJE. OGSAA VASK
MOV(021) &0 L1_2_SPERR_KODE_INN
; rung 1: B0111  TEMP INN TIL KJØLER
LD P_On
/F(457) B0111_TT DIVISOR_INNGANGSORD B0111_HJREG1  ; ZZ, DELER INGANGSVERDI MED 32,760 FOR OMREGNING TIL 0-1000
FIX(450) B0111_HJREG1 B0111_0_1000  ; 0=0GRADER   1000=100.0 GRADER

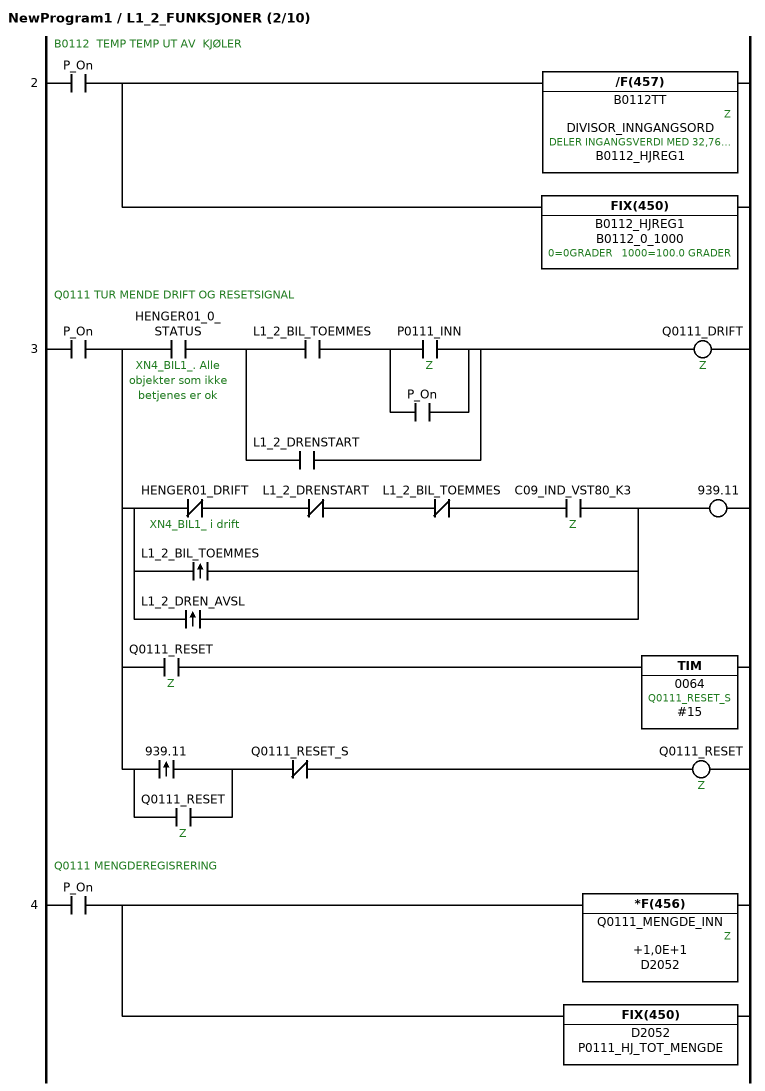
; rung 2: B0112  TEMP TEMP UT AV  KJØLER
LD P_On
/F(457) B0112TT DIVISOR_INNGANGSORD B0112_HJREG1  ; Z, DELER INGANGSVERDI MED 32,760 FOR OMREGNING TIL 0-1000
FIX(450) B0112_HJREG1 B0112_0_1000  ; 0=0GRADER   1000=100.0 GRADER
; rung 3: Q0111 TUR MENDE DRIFT OG RESETSIGNAL
LD P_On
OUT TR0
AND HENGER01_0_STATUS  ; XN4_BIL1_. Alle objekter som ikke betjenes er ok
LD L1_2_BIL_TOEMMES
LD P0111_INN  ; Z
OR P_On
ANDLD
OR L1_2_DRENSTART
ANDLD
OUT Q0111_DRIFT  ; Z
LD TR0
LDNOT HENGER01_DRIFT  ; XN4_BIL1_ i drift
ANDNOT L1_2_DRENSTART
ANDNOT L1_2_BIL_TOEMMES
AND C09_IND_VST80_K3  ; Z
@OR L1_2_BIL_TOEMMES
@OR L1_2_DREN_AVSL
ANDLD
OUT 939.11
LD TR0
AND Q0111_RESET  ; Z
TIM 0064 #15  ; Q0111_RESET_S
LD TR0
@LD 939.11
OR Q0111_RESET  ; Z
ANDLD
ANDNOT Q0111_RESET_S
OUT Q0111_RESET  ; Z
; rung 4: Q0111 MENGDEREGISRERING
LD P_On
*F(456) Q0111_MENGDE_INN +1,0E+1 D2052  ; Z
FIX(450) D2052 P0111_HJ_TOT_MENGDE

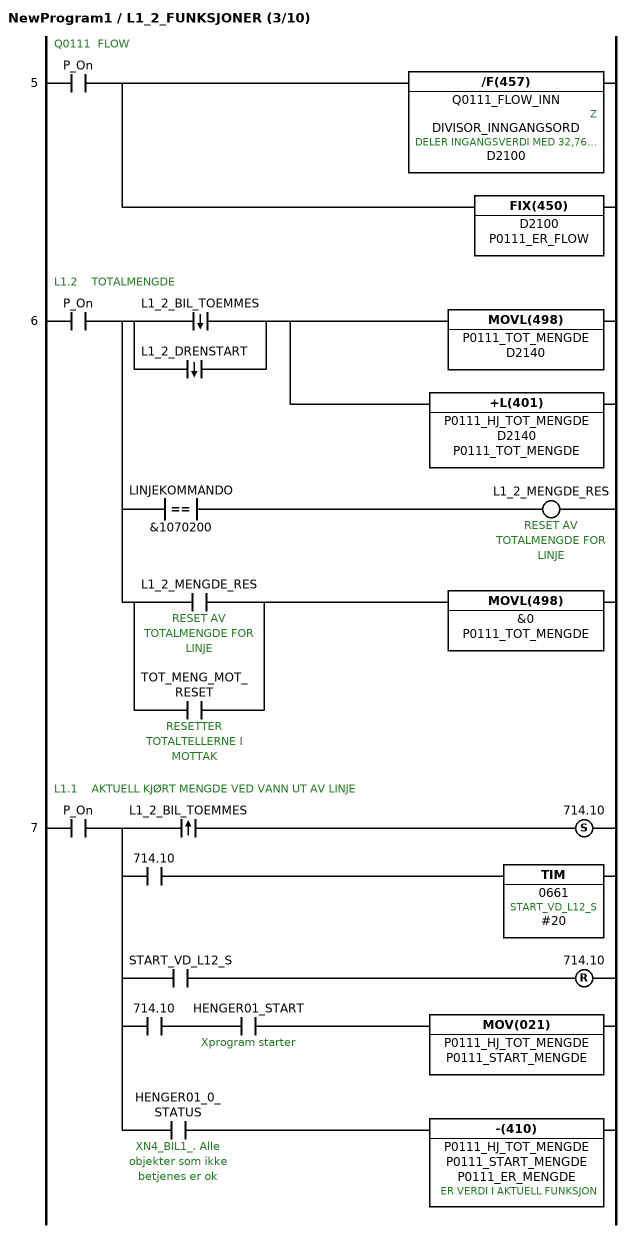
; rung 5: Q0111  FLOW
LD P_On
/F(457) Q0111_FLOW_INN DIVISOR_INNGANGSORD D2100  ; Z, DELER INGANGSVERDI MED 32,760 FOR OMREGNING TIL 0-1000
FIX(450) D2100 P0111_ER_FLOW
; rung 6: L1.2    TOTALMENGDE
LD P_On
OUT TR0
%LD L1_2_BIL_TOEMMES
%OR L1_2_DRENSTART
ANDLD
MOVL(498) P0111_TOT_MENGDE D2140
+L(401) P0111_HJ_TOT_MENGDE D2140 P0111_TOT_MENGDE
LD TR0
AND=L(301) LINJEKOMMANDO &1070200
OUT L1_2_MENGDE_RES  ; RESET AV  TOTALMENGDE FOR LINJE
LD TR0
LD L1_2_MENGDE_RES  ; RESET AV  TOTALMENGDE FOR LINJE
OR TOT_MENG_MOT_RESET  ; RESETTER TOTALTELLERNE I MOTTAK
ANDLD
MOVL(498) &0 P0111_TOT_MENGDE
; rung 7: L1.1    AKTUELL KJØRT MENGDE VED VANN UT AV LINJE
LD P_On
OUT TR0
@AND L1_2_BIL_TOEMMES
SET 714.10
LD TR0
AND 714.10
TIM 0661 #20  ; START_VD_L12_S
LD TR0
AND START_VD_L12_S
RSET 714.10
LD TR0
AND 714.10
AND HENGER01_START  ; Xprogram starter
MOV(021) P0111_HJ_TOT_MENGDE P0111_START_MENGDE
LD TR0
AND HENGER01_0_STATUS  ; XN4_BIL1_. Alle objekter som ikke betjenes er ok
-(410) P0111_HJ_TOT_MENGDE P0111_START_MENGDE P0111_ER_MENGDE  ; ER VERDI I AKTUELL FUNKSJON

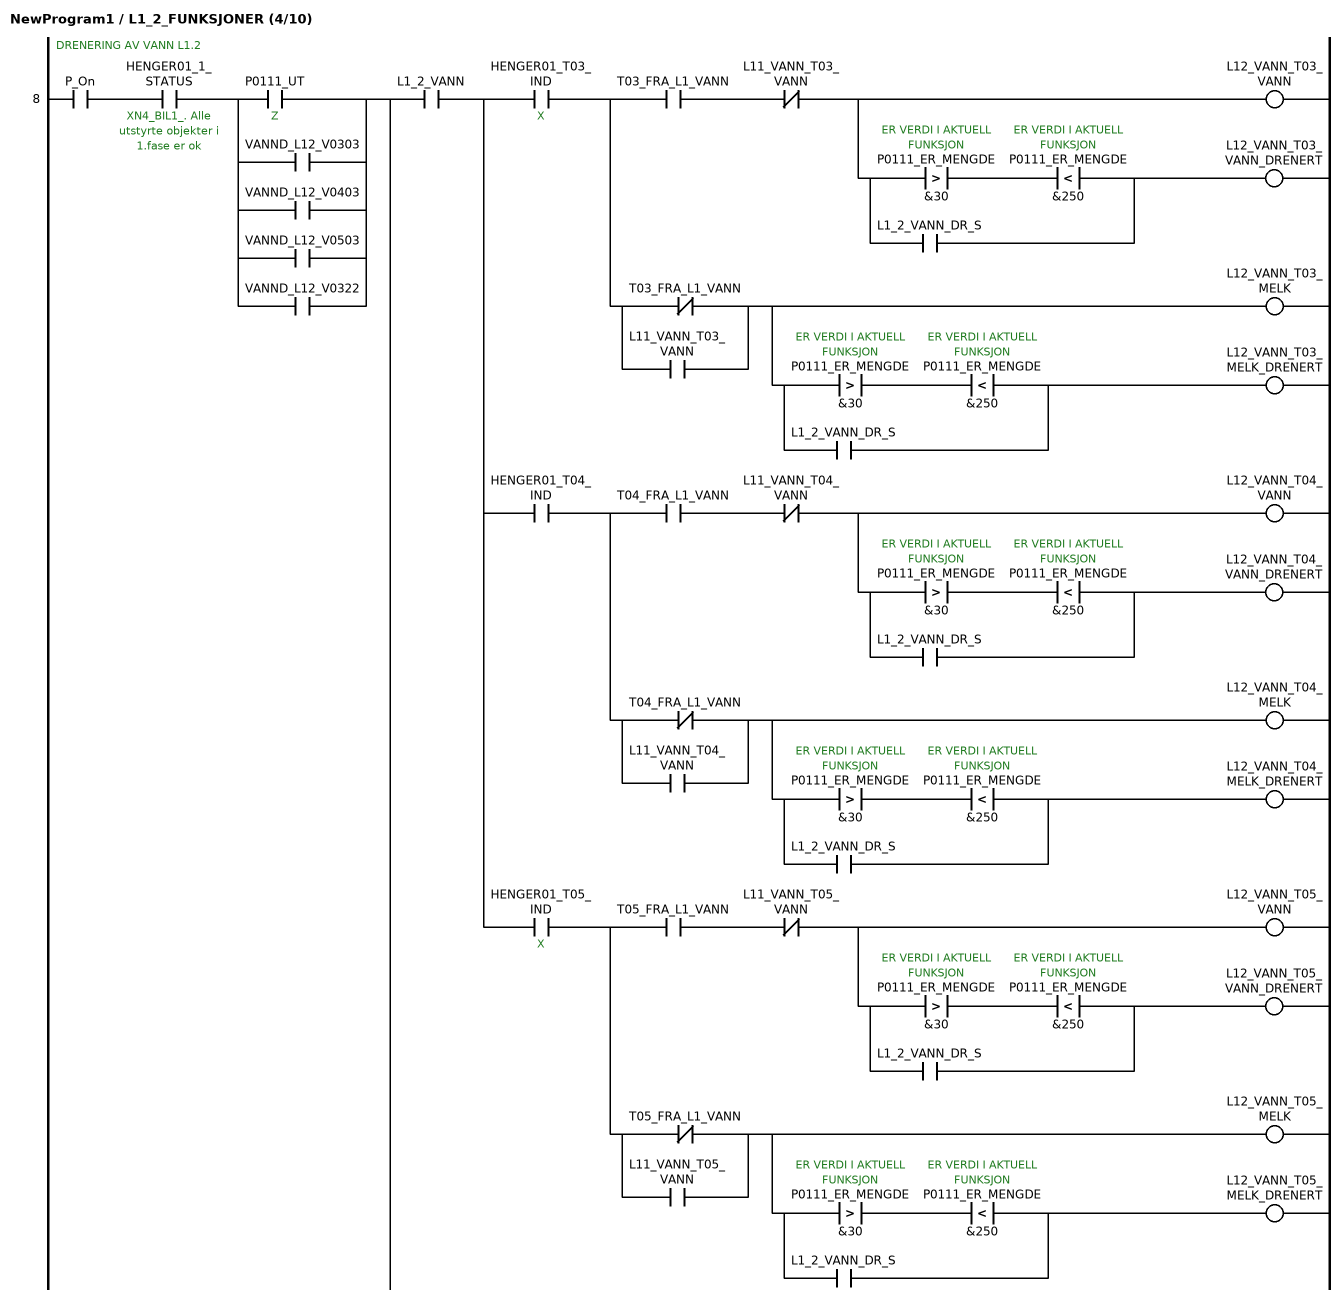

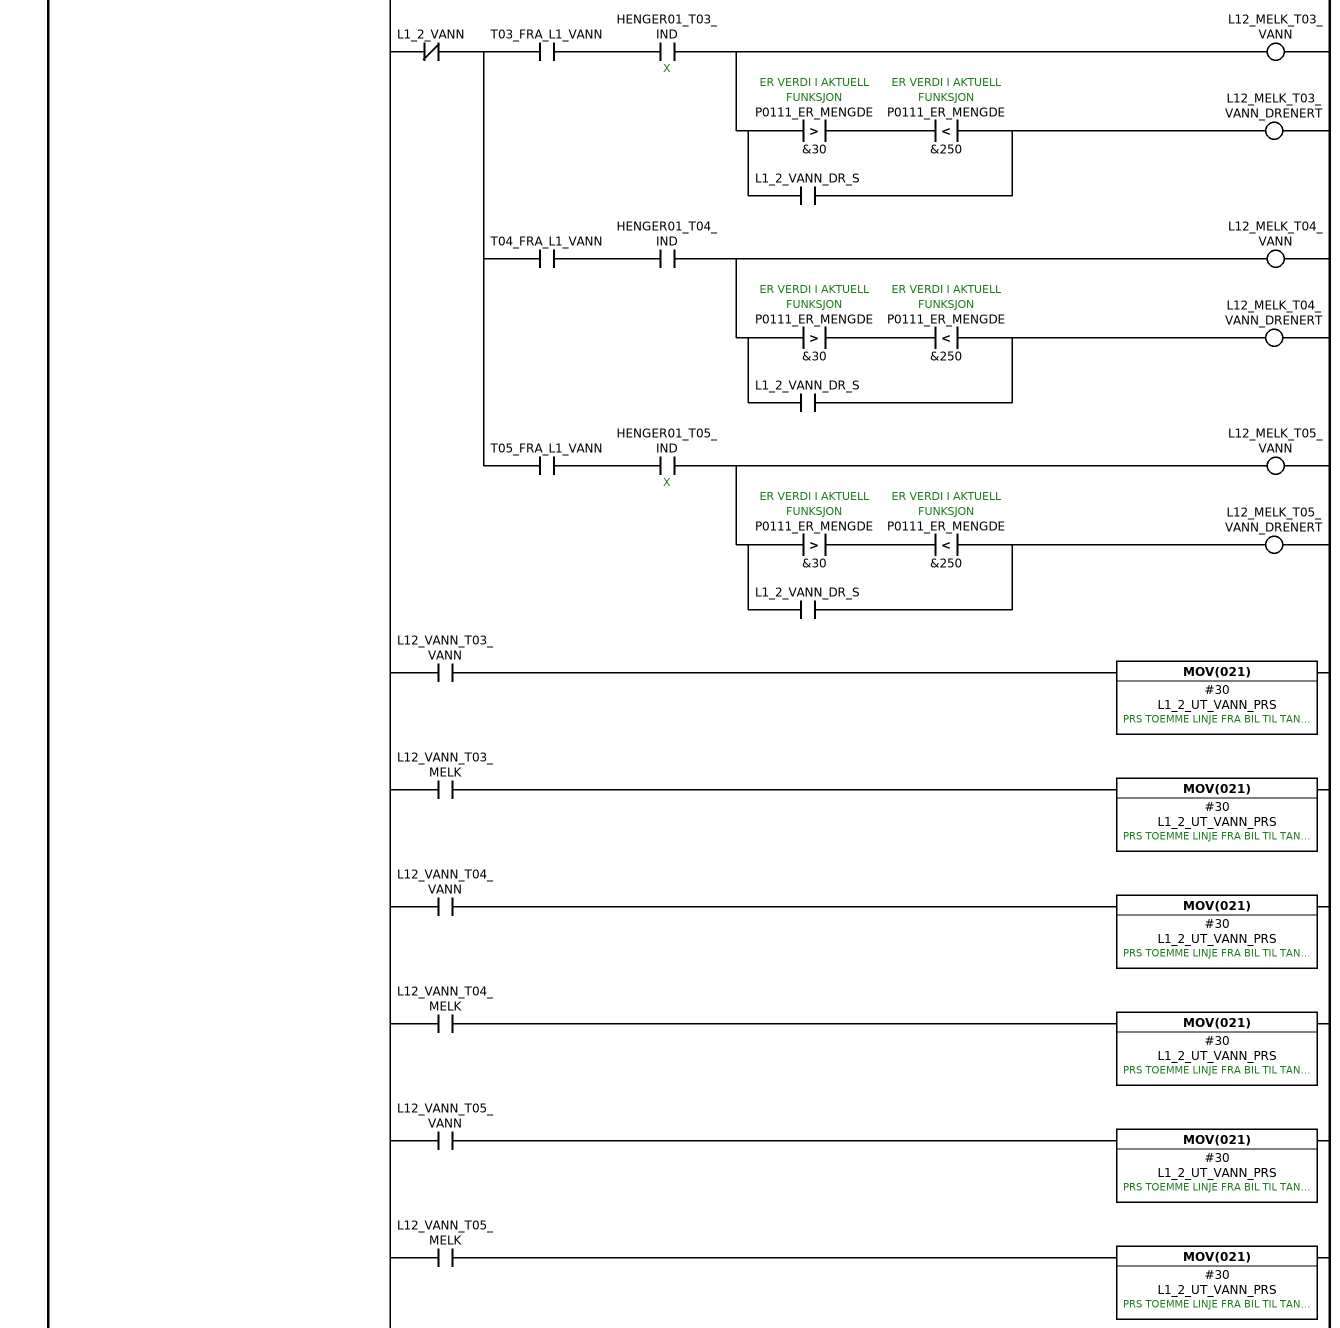

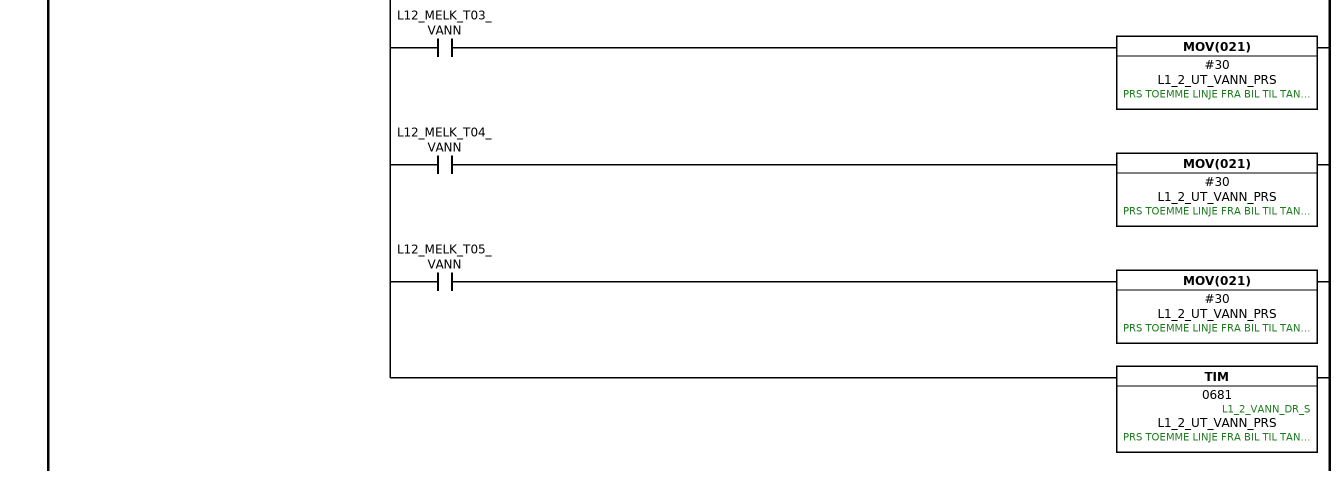
; rung 8: DRENERING AV VANN L1.2
LD P_On
AND HENGER01_1_STATUS  ; XN4_BIL1_. Alle utstyrte objekter i 1.fase er ok
LD P0111_UT  ; Z
OR VANND_L12_V0303
OR VANND_L12_V0403
OR VANND_L12_V0503
OR VANND_L12_V0322
ANDLD
OUT TR0
AND L1_2_VANN
OUT TR1
AND HENGER01_T03_IND  ; X
OUT TR2
AND T03_FRA_L1_VANN
ANDNOT L11_VANN_T03_VANN
OUT L12_VANN_T03_VANN
LD>(320) P0111_ER_MENGDE &30  ; ER VERDI I AKTUELL FUNKSJON
AND<(310) P0111_ER_MENGDE &250  ; ER VERDI I AKTUELL FUNKSJON
OR L1_2_VANN_DR_S
ANDLD
OUT L12_VANN_T03_VANN_DRENERT
LD TR2
LDNOT T03_FRA_L1_VANN
OR L11_VANN_T03_VANN
ANDLD
OUT L12_VANN_T03_MELK
LD>(320) P0111_ER_MENGDE &30  ; ER VERDI I AKTUELL FUNKSJON
AND<(310) P0111_ER_MENGDE &250  ; ER VERDI I AKTUELL FUNKSJON
OR L1_2_VANN_DR_S
ANDLD
OUT L12_VANN_T03_MELK_DRENERT
LD TR1
AND HENGER01_T04_IND
OUT TR2
AND T04_FRA_L1_VANN
ANDNOT L11_VANN_T04_VANN
OUT L12_VANN_T04_VANN
LD>(320) P0111_ER_MENGDE &30  ; ER VERDI I AKTUELL FUNKSJON
AND<(310) P0111_ER_MENGDE &250  ; ER VERDI I AKTUELL FUNKSJON
OR L1_2_VANN_DR_S
ANDLD
OUT L12_VANN_T04_VANN_DRENERT
LD TR2
LDNOT T04_FRA_L1_VANN
OR L11_VANN_T04_VANN
ANDLD
OUT L12_VANN_T04_MELK
LD>(320) P0111_ER_MENGDE &30  ; ER VERDI I AKTUELL FUNKSJON
AND<(310) P0111_ER_MENGDE &250  ; ER VERDI I AKTUELL FUNKSJON
OR L1_2_VANN_DR_S
ANDLD
OUT L12_VANN_T04_MELK_DRENERT
LD TR1
AND HENGER01_T05_IND  ; X
OUT TR1
AND T05_FRA_L1_VANN
ANDNOT L11_VANN_T05_VANN
OUT L12_VANN_T05_VANN
LD>(320) P0111_ER_MENGDE &30  ; ER VERDI I AKTUELL FUNKSJON
AND<(310) P0111_ER_MENGDE &250  ; ER VERDI I AKTUELL FUNKSJON
OR L1_2_VANN_DR_S
ANDLD
OUT L12_VANN_T05_VANN_DRENERT
LD TR1
LDNOT T05_FRA_L1_VANN
OR L11_VANN_T05_VANN
ANDLD
OUT L12_VANN_T05_MELK
LD>(320) P0111_ER_MENGDE &30  ; ER VERDI I AKTUELL FUNKSJON
AND<(310) P0111_ER_MENGDE &250  ; ER VERDI I AKTUELL FUNKSJON
OR L1_2_VANN_DR_S
ANDLD
OUT L12_VANN_T05_MELK_DRENERT
LD TR0
ANDNOT L1_2_VANN
OUT TR1
AND T03_FRA_L1_VANN
AND HENGER01_T03_IND  ; X
OUT L12_MELK_T03_VANN
LD>(320) P0111_ER_MENGDE &30  ; ER VERDI I AKTUELL FUNKSJON
AND<(310) P0111_ER_MENGDE &250  ; ER VERDI I AKTUELL FUNKSJON
OR L1_2_VANN_DR_S
ANDLD
OUT L12_MELK_T03_VANN_DRENERT
LD TR1
AND T04_FRA_L1_VANN
AND HENGER01_T04_IND
OUT L12_MELK_T04_VANN
LD>(320) P0111_ER_MENGDE &30  ; ER VERDI I AKTUELL FUNKSJON
AND<(310) P0111_ER_MENGDE &250  ; ER VERDI I AKTUELL FUNKSJON
OR L1_2_VANN_DR_S
ANDLD
OUT L12_MELK_T04_VANN_DRENERT
LD TR1
AND T05_FRA_L1_VANN
AND HENGER01_T05_IND  ; X
OUT L12_MELK_T05_VANN
LD>(320) P0111_ER_MENGDE &30  ; ER VERDI I AKTUELL FUNKSJON
AND<(310) P0111_ER_MENGDE &250  ; ER VERDI I AKTUELL FUNKSJON
OR L1_2_VANN_DR_S
ANDLD
OUT L12_MELK_T05_VANN_DRENERT
LD TR0
AND L12_VANN_T03_VANN
MOV(021) #30 L1_2_UT_VANN_PRS  ; PRS TOEMME LINJE FRA BIL TIL TANK FOR VANN
LD TR0
AND L12_VANN_T03_MELK
MOV(021) #30 L1_2_UT_VANN_PRS  ; PRS TOEMME LINJE FRA BIL TIL TANK FOR VANN
LD TR0
AND L12_VANN_T04_VANN
MOV(021) #30 L1_2_UT_VANN_PRS  ; PRS TOEMME LINJE FRA BIL TIL TANK FOR VANN
LD TR0
AND L12_VANN_T04_MELK
MOV(021) #30 L1_2_UT_VANN_PRS  ; PRS TOEMME LINJE FRA BIL TIL TANK FOR VANN
LD TR0
AND L12_VANN_T05_VANN
MOV(021) #30 L1_2_UT_VANN_PRS  ; PRS TOEMME LINJE FRA BIL TIL TANK FOR VANN
LD TR0
AND L12_VANN_T05_MELK
MOV(021) #30 L1_2_UT_VANN_PRS  ; PRS TOEMME LINJE FRA BIL TIL TANK FOR VANN
LD TR0
AND L12_MELK_T03_VANN
MOV(021) #30 L1_2_UT_VANN_PRS  ; PRS TOEMME LINJE FRA BIL TIL TANK FOR VANN
LD TR0
AND L12_MELK_T04_VANN
MOV(021) #30 L1_2_UT_VANN_PRS  ; PRS TOEMME LINJE FRA BIL TIL TANK FOR VANN
LD TR0
AND L12_MELK_T05_VANN
MOV(021) #30 L1_2_UT_VANN_PRS  ; PRS TOEMME LINJE FRA BIL TIL TANK FOR VANN
LD TR0
TIM 0681 L1_2_UT_VANN_PRS  ; PRS TOEMME LINJE FRA BIL TIL TANK FOR VANN, L1_2_VANN_DR_S

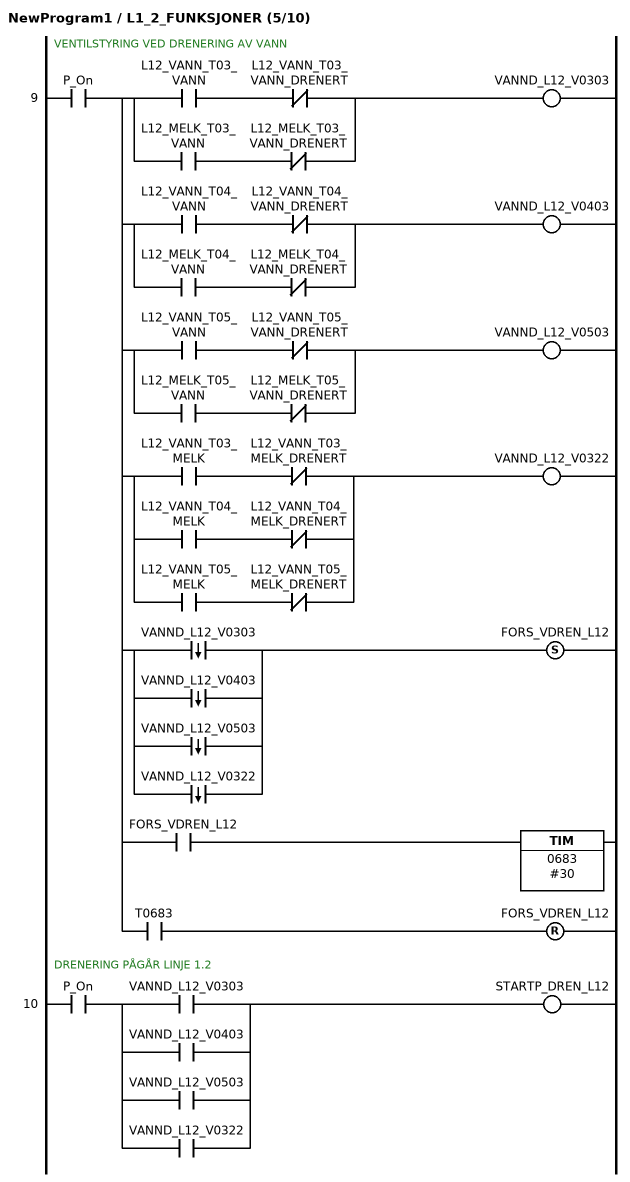
; rung 9: VENTILSTYRING VED DRENERING AV VANN
LD P_On
OUT TR0
LD L12_VANN_T03_VANN
ANDNOT L12_VANN_T03_VANN_DRENERT
LD L12_MELK_T03_VANN
ANDNOT L12_MELK_T03_VANN_DRENERT
ORLD
ANDLD
OUT VANND_L12_V0303
LD TR0
LD L12_VANN_T04_VANN
ANDNOT L12_VANN_T04_VANN_DRENERT
LD L12_MELK_T04_VANN
ANDNOT L12_MELK_T04_VANN_DRENERT
ORLD
ANDLD
OUT VANND_L12_V0403
LD TR0
LD L12_VANN_T05_VANN
ANDNOT L12_VANN_T05_VANN_DRENERT
LD L12_MELK_T05_VANN
ANDNOT L12_MELK_T05_VANN_DRENERT
ORLD
ANDLD
OUT VANND_L12_V0503
LD TR0
LD L12_VANN_T03_MELK
ANDNOT L12_VANN_T03_MELK_DRENERT
LD L12_VANN_T04_MELK
ANDNOT L12_VANN_T04_MELK_DRENERT
ORLD
LD L12_VANN_T05_MELK
ANDNOT L12_VANN_T05_MELK_DRENERT
ORLD
ANDLD
OUT VANND_L12_V0322
LD TR0
%LD VANND_L12_V0303
%OR VANND_L12_V0403
%OR VANND_L12_V0503
%OR VANND_L12_V0322
ANDLD
SET FORS_VDREN_L12
LD TR0
AND FORS_VDREN_L12
TIM 0683 #30
LD TR0
AND T0683
RSET FORS_VDREN_L12
; rung 10: DRENERING PÅGÅR LINJE 1.2
LD P_On
LD VANND_L12_V0303
OR VANND_L12_V0403
OR VANND_L12_V0503
OR VANND_L12_V0322
ANDLD
OUT STARTP_DREN_L12

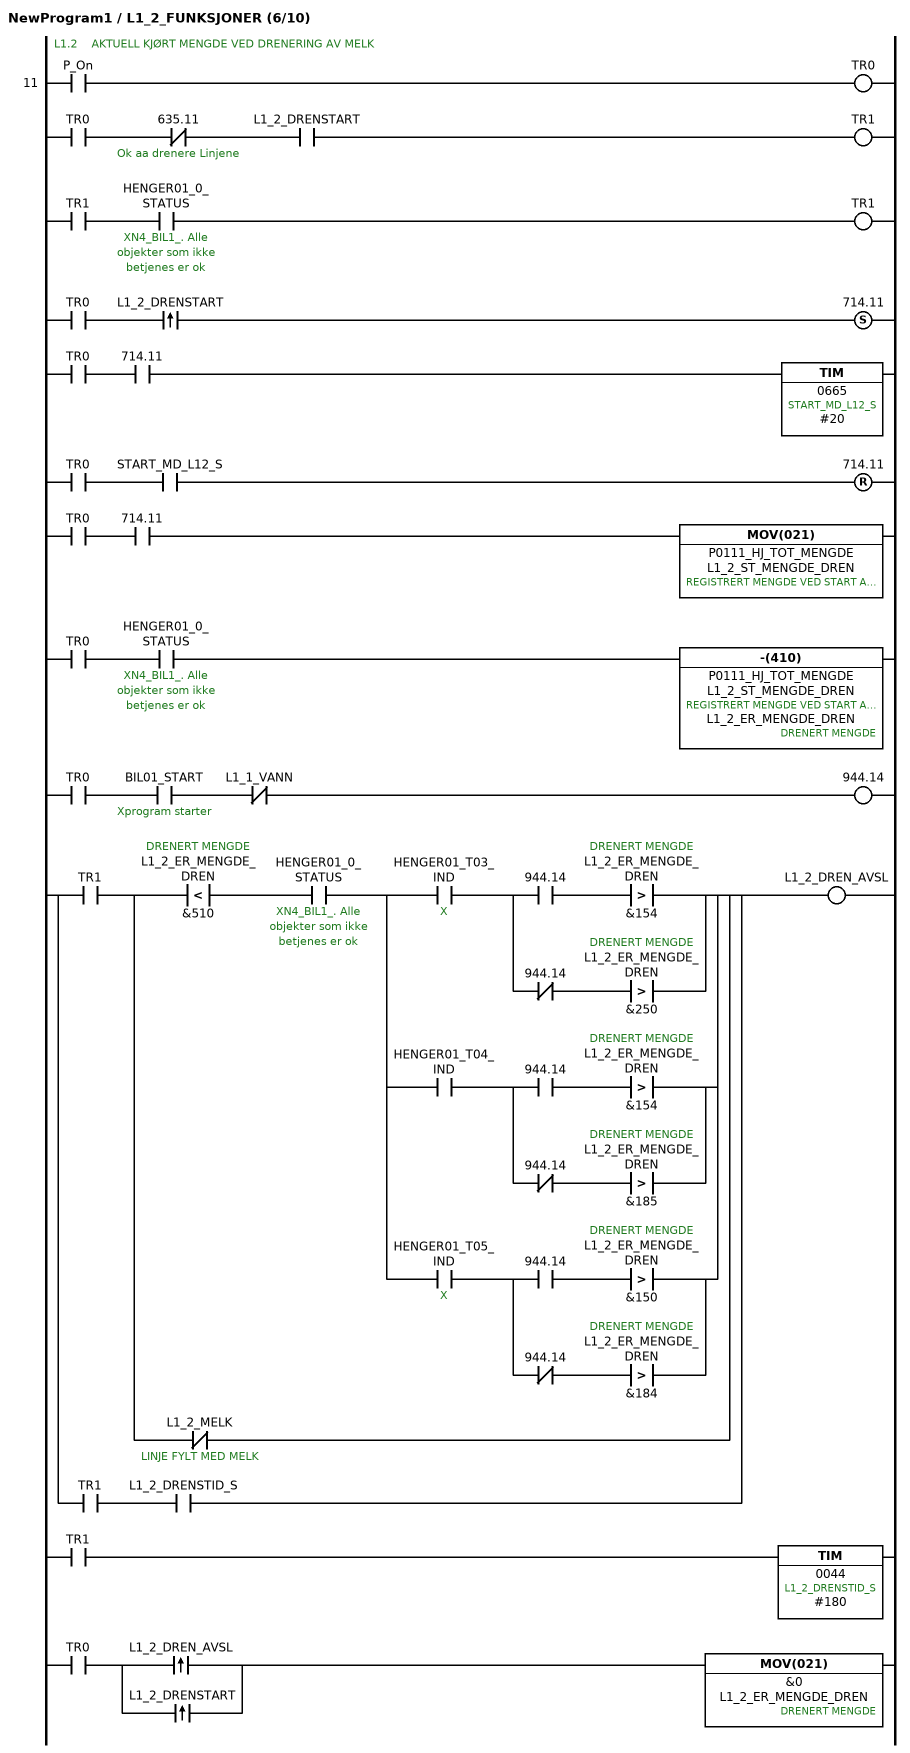
; rung 11: L1.2    AKTUELL KJØRT MENGDE VED DRENERING AV MELK
LD P_On
OUT TR0
@AND L1_2_DRENSTART
SET 714.11
LD TR0
AND 714.11
TIM 0665 #20  ; START_MD_L12_S
LD TR0
AND START_MD_L12_S
RSET 714.11
LD TR0
AND 714.11
MOV(021) P0111_HJ_TOT_MENGDE L1_2_ST_MENGDE_DREN  ; REGISTRERT MENGDE VED START AV DREN.
LD TR0
AND HENGER01_0_STATUS  ; XN4_BIL1_. Alle objekter som ikke betjenes er ok
-(410) P0111_HJ_TOT_MENGDE L1_2_ST_MENGDE_DREN L1_2_ER_MENGDE_DREN  ; REGISTRERT MENGDE VED START AV DREN., DRENERT MENGDE
LD TR0
AND BIL01_START  ; Xprogram starter
ANDNOT L1_1_VANN
OUT 944.14
LD TR0
ANDNOT 635.11  ; Ok aa drenere Linjene
AND L1_2_DRENSTART
OUT TR1
LD<(310) L1_2_ER_MENGDE_DREN &510  ; DRENERT MENGDE
AND HENGER01_0_STATUS  ; XN4_BIL1_. Alle objekter som ikke betjenes er ok
LD HENGER01_T03_IND  ; X
LD 944.14
AND>(320) L1_2_ER_MENGDE_DREN &154  ; DRENERT MENGDE
LDNOT 944.14
AND>(320) L1_2_ER_MENGDE_DREN &250  ; DRENERT MENGDE
ORLD
ANDLD
LD HENGER01_T04_IND
LD 944.14
AND>(320) L1_2_ER_MENGDE_DREN &154  ; DRENERT MENGDE
LDNOT 944.14
AND>(320) L1_2_ER_MENGDE_DREN &185  ; DRENERT MENGDE
ORLD
ANDLD
ORLD
LD HENGER01_T05_IND  ; X
LD 944.14
AND>(320) L1_2_ER_MENGDE_DREN &150  ; DRENERT MENGDE
LDNOT 944.14
AND>(320) L1_2_ER_MENGDE_DREN &184  ; DRENERT MENGDE
ORLD
ANDLD
ORLD
ANDLD
ORNOT L1_2_MELK  ; LINJE FYLT MED MELK
ANDLD
LD TR1
AND HENGER01_0_STATUS  ; XN4_BIL1_. Alle objekter som ikke betjenes er ok
OUT TR1
AND L1_2_DRENSTID_S
ORLD
OUT L1_2_DREN_AVSL
LD TR1
TIM 0044 #180  ; L1_2_DRENSTID_S
LD TR0
@LD L1_2_DREN_AVSL
@OR L1_2_DRENSTART
ANDLD
MOV(021) &0 L1_2_ER_MENGDE_DREN  ; DRENERT MENGDE

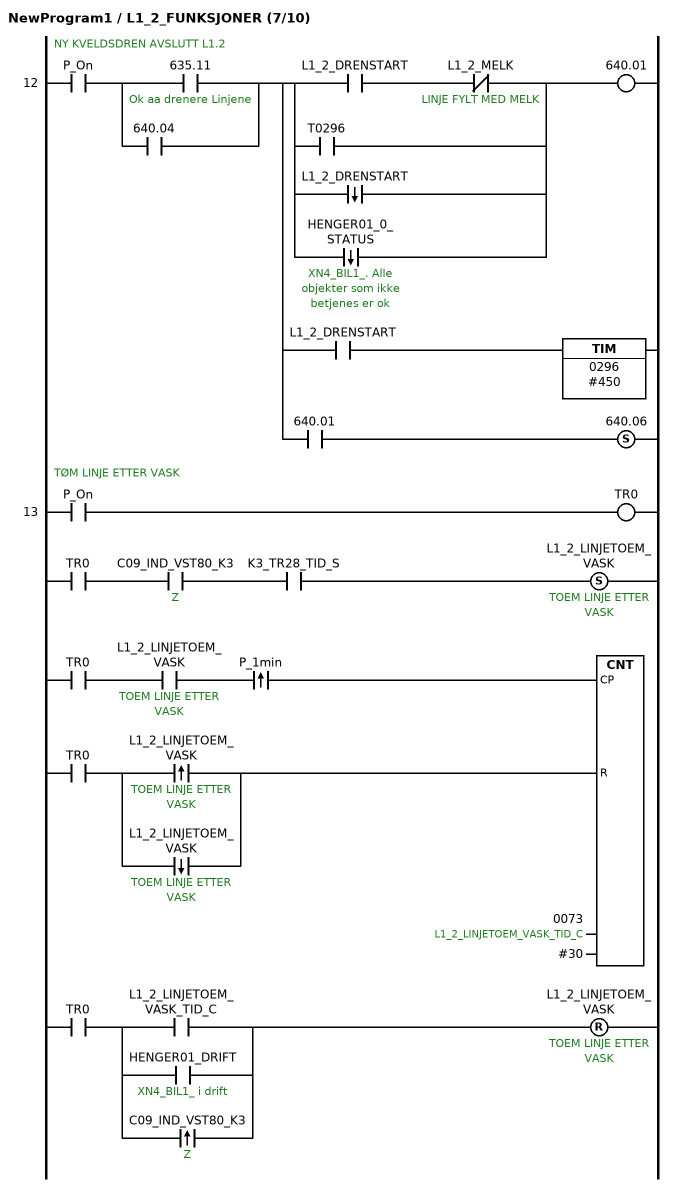
; rung 12: NY KVELDSDREN AVSLUTT L1.2
LD P_On
LD 635.11  ; Ok aa drenere Linjene
OR 640.04
ANDLD
OUT TR0
LD L1_2_DRENSTART
ANDNOT L1_2_MELK  ; LINJE FYLT MED MELK
OR T0296
%OR L1_2_DRENSTART
%OR HENGER01_0_STATUS  ; XN4_BIL1_. Alle objekter som ikke betjenes er ok
ANDLD
OUT 640.01
LD TR0
AND L1_2_DRENSTART
TIM 0296 #450
LD TR0
AND 640.01
SET 640.06
; rung 13: TØM LINJE ETTER VASK
LD P_On
OUT TR0
AND C09_IND_VST80_K3  ; Z
AND K3_TR28_TID_S
SET L1_2_LINJETOEM_VASK  ; TOEM LINJE ETTER VASK
LD TR0
AND L1_2_LINJETOEM_VASK  ; TOEM LINJE ETTER VASK
@AND P_1min
LD TR0
@LD L1_2_LINJETOEM_VASK  ; TOEM LINJE ETTER VASK
%OR L1_2_LINJETOEM_VASK  ; TOEM LINJE ETTER VASK
ANDLD
CNT 0073 #30  ; L1_2_LINJETOEM_VASK_TID_C
LD TR0
LD L1_2_LINJETOEM_VASK_TID_C
OR HENGER01_DRIFT  ; XN4_BIL1_ i drift
@OR C09_IND_VST80_K3  ; Z
ANDLD
RSET L1_2_LINJETOEM_VASK  ; TOEM LINJE ETTER VASK

